LIN {X 0,Y 299.694,Z 797.286,A -85,B 0,C 180,E1 14832.527,E2 14832.527} C_VEL
LIN {X 0,Y 302.392,Z 789.527,A -85,B 0,C 180,E1 14828.672,E2 14828.672} C_VEL
LIN {X 0,Y 305.884,Z 780.362,A -85,B 0,C 180,E1 14825.061,E2 14825.061} C_VEL
LIN {X 0,Y 310.162,Z 769.656,A -85,B 0,C 180,E1 14821.65,E2 14821.65} C_VEL
LIN {X 0,Y 315.139,Z 757.152,A -85,B 0,C 180,E1 14818.433,E2 14818.433} C_VEL
LIN {X 0,Y 319.478,Z 746.033,A -85,B 0,C 180,E1 14816.053,E2 14816.053} C_VEL
LIN {X 0,Y 320.57,Z 741.155,A -85,B 0,C 180,E1 14814.994,E2 14814.994} C_VEL
LIN {X 0,Y 320.588,Z 728.797,A -85,B 0,C 180,E1 14812.148,E2 14812.148} C_VEL
LIN {X 0,Y 321.792,Z 723.281,A -85,B 0,C 180,E1 14811.202,E2 14811.202} C_VEL
LIN {X 0,Y 327.57,Z 706.668,A -85,B 0,C 180,E1 14808.986,E2 14808.986} C_VEL
LIN {X 0,Y 332.904,Z 689.548,A -85,B 0,C 180,E1 14807.126,E2 14807.126} C_VEL
LIN {X 0,Y 338.125,Z 670.498,A -85,B 0,C 180,E1 14805.452,E2 14805.452} C_VEL
LIN {X 0,Y 342.569,Z 651.293,A -85,B 0,C 180,E1 14804.112,E2 14804.112} C_VEL
LIN {X 0,Y 346.403,Z 631.027,A -85,B 0,C 180,E1 14803.025,E2 14803.025} C_VEL
LIN {X 0,Y 349.317,Z 610.319,A -85,B 0,C 180,E1 14802.217,E2 14802.217} C_VEL
LIN {X 0,Y 351.212,Z 589.58,A -85,B 0,C 180,E1 14801.664,E2 14801.664} C_VEL
LIN {X 0,Y 361.538,Z 397.142,A -85,B 0,C 180,E1 14797.851,E2 14797.851} C_VEL
LIN {X 0,Y 353.208,Z 382.377,A -85,B 0,C 180,E1 14795.383,E2 14795.383} C_VEL
LIN {X 0,Y 344.318,Z 367.821,A -85,B 0,C 180,E1 14792.446,E2 14792.446} C_VEL
LIN {X 0,Y 335.968,Z 355.363,A -85,B 0,C 180,E1 14789.313,E2 14789.313} C_VEL
LIN {X 0,Y 329.419,Z 346.302,A -85,B 0,C 180,E1 14786.499,E2 14786.499} C_VEL
LIN {X 0,Y 325.161,Z 340.597,A -85,B 0,C 180,E1 14784.43,E2 14784.43} C_VEL
LIN {X 0,Y 321.712,Z 336.158,A -85,B 0,C 180,E1 14782.571,E2 14782.571} C_VEL
LIN {X 0,Y 318.302,Z 331.619,A -85,B 0,C 180,E1 14780.503,E2 14780.503} C_VEL
LIN {X 0,Y 314.842,Z 327.176,A -85,B 0,C 180,E1 14778.085,E2 14778.085} C_VEL
LIN {X 0,Y 309.683,Z 320.807,A -85,B 0,C 180,E1 14773.442,E2 14773.442} C_VEL
LIN {X 0,Y 305.683,Z 315.348,A -85,B 0,C 180,E1 14766.197,E2 14766.197} C_VEL
LIN {X 0,Y 305.143,Z 314.738,A -85,B 0,C 180,E1 14761.127,E2 14761.127} C_VEL
LIN {X 0,Y 306.221,Z 315.739,A -85,B 0,C 180,E1 14756.818,E2 14756.818} C_VEL
LIN {X 0,Y 312.094,Z 322.032,A -85,B 0,C 180,E1 14749.385,E2 14749.385} C_VEL
LIN {X 0,Y 315.714,Z 326.528,A -85,B 0,C 180,E1 14746.447,E2 14746.447} C_VEL
LIN {X 0,Y 317.507,Z 328.292,A -85,B 0,C 180,E1 14745.222,E2 14745.222} C_VEL
LIN {X 0,Y 321.089,Z 332.723,A -85,B 0,C 180,E1 14742.98,E2 14742.98} C_VEL
LIN {X 0,Y 322.59,Z 334.467,A -85,B 0,C 180,E1 14742.131,E2 14742.131} C_VEL
LIN {X 0,Y 327.326,Z 340.382,A -85,B 0,C 180,E1 14739.668,E2 14739.668} C_VEL
LIN {X 0,Y 334.059,Z 349.029,A -85,B 0,C 180,E1 14736.636,E2 14736.636} C_VEL
LIN {X 0,Y 341.6,Z 359.524,A -85,B 0,C 180,E1 14733.677,E2 14733.677} C_VEL
LIN {X 0,Y 349.604,Z 371.289,A -85,B 0,C 180,E1 14730.91,E2 14730.91} C_VEL
LIN {X 0,Y 358.032,Z 384.909,A -85,B 0,C 180,E1 14728.284,E2 14728.284} C_VEL
LIN {X 0,Y 363.686,Z 394.863,A -85,B 0,C 180,E1 14726.65,E2 14726.65} C_VEL
LIN {X 0,Y 351.066,Z 599.637,A -85,B 0,C 180,E1 14722.328,E2 14722.328} C_VEL
LIN {X 0,Y 348.542,Z 622.55,A -85,B 0,C 180,E1 14721.656,E2 14721.656} C_VEL
LIN {X 0,Y 345.195,Z 643.809,A -85,B 0,C 180,E1 14720.786,E2 14720.786} C_VEL
LIN {X 0,Y 341.362,Z 663.255,A -85,B 0,C 180,E1 14719.728,E2 14719.728} C_VEL
LIN {X 0,Y 336.622,Z 683.448,A -85,B 0,C 180,E1 14718.331,E2 14718.331} C_VEL
LIN {X 0,Y 331.361,Z 702.998,A -85,B 0,C 180,E1 14716.65,E2 14716.65} C_VEL
LIN {X 0,Y 325.719,Z 721.816,A -85,B 0,C 180,E1 14714.663,E2 14714.663} C_VEL
LIN {X 0,Y 319.825,Z 739.772,A -85,B 0,C 180,E1 14712.333,E2 14712.333} C_VEL
LIN {X 0,Y 313.923,Z 756.677,A -85,B 0,C 180,E1 14709.686,E2 14709.686} C_VEL
LIN {X 0,Y 308.396,Z 772.066,A -85,B 0,C 180,E1 14706.794,E2 14706.794} C_VEL
LIN {X 0,Y 303.032,Z 786.885,A -85,B 0,C 180,E1 14703.436,E2 14703.436} C_VEL
LIN {X 0,Y 298.504,Z 799.576,A -85,B 0,C 180,E1 14699.939,E2 14699.939} C_VEL
LIN {X 0,Y 294.718,Z 810.947,A -85,B 0,C 180,E1 14696.169,E2 14696.169} C_VEL
LIN {X 0,Y 291.911,Z 820.502,A -85,B 0,C 180,E1 14692.345,E2 14692.345} C_VEL
LIN {X 0,Y 289.889,Z 828.607,A -85,B 0,C 180,E1 14688.292,E2 14688.292} C_VEL
LIN {X 0,Y 288.661,Z 835.273,A -85,B 0,C 180,E1 14684.032,E2 14684.032} C_VEL
LIN {X 0,Y 288.163,Z 840.012,A -85,B 0,C 180,E1 14679.99,E2 14679.99} C_VEL
LIN {X 0,Y 288.063,Z 842.936,A -85,B 0,C 180,E1 14676.177,E2 14676.177} C_VEL
LIN {X 0,Y 288.1,Z 844.57,A -85,B 0,C 180,E1 14672.387,E2 14672.387} C_VEL
LIN {X 0,Y 288.115,Z 844.72,A -85,B 0,C 180,E1 14668.807,E2 14668.807} C_VEL
LIN {X 0,Y 288.075,Z 843.64,A -85,B 0,C 180,E1 14665.022,E2 14665.022} C_VEL
LIN {X 0,Y 288.102,Z 841.035,A -85,B 0,C 180,E1 14661.217,E2 14661.217} C_VEL
LIN {X 0,Y 288.456,Z 836.889,A -85,B 0,C 180,E1 14657.183,E2 14657.183} C_VEL
LIN {X 0,Y 289.385,Z 831.018,A -85,B 0,C 180,E1 14653.129,E2 14653.129} C_VEL
LIN {X 0,Y 291.195,Z 823.048,A -85,B 0,C 180,E1 14648.868,E2 14648.868} C_VEL
LIN {X 0,Y 293.882,Z 813.618,A -85,B 0,C 180,E1 14644.832,E2 14644.832} C_VEL
LIN {X 0,Y 297.621,Z 802.16,A -85,B 0,C 180,E1 14640.849,E2 14640.849} C_VEL
LIN {X 0,Y 302.108,Z 789.305,A -85,B 0,C 180,E1 14637.207,E2 14637.207} C_VEL
LIN {X 0,Y 307.183,Z 775.278,A -85,B 0,C 180,E1 14633.905,E2 14633.905} C_VEL
LIN {X 0,Y 312.801,Z 759.732,A -85,B 0,C 180,E1 14630.855,E2 14630.855} C_VEL
LIN {X 0,Y 318.644,Z 743.198,A -85,B 0,C 180,E1 14628.168,E2 14628.168} C_VEL
LIN {X 0,Y 324.354,Z 725.842,A -85,B 0,C 180,E1 14625.841,E2 14625.841} C_VEL
LIN {X 0,Y 330.137,Z 706.989,A -85,B 0,C 180,E1 14623.755,E2 14623.755} C_VEL
LIN {X 0,Y 335.514,Z 687.59,A -85,B 0,C 180,E1 14622,E2 14622} C_VEL
LIN {X 0,Y 340.548,Z 666.776,A -85,B 0,C 180,E1 14620.5,E2 14620.5} C_VEL
LIN {X 0,Y 344.609,Z 646.553,A -85,B 0,C 180,E1 14619.362,E2 14619.362} C_VEL
LIN {X 0,Y 348.2,Z 624.526,A -85,B 0,C 180,E1 14618.425,E2 14618.425} C_VEL
LIN {X 0,Y 350.748,Z 602.835,A -85,B 0,C 180,E1 14617.76,E2 14617.76} C_VEL
LIN {X 0,Y 362.34,Z 415.076,A -85,B 0,C 180,E1 14613.778,E2 14613.778} C_VEL
LIN {X 0,Y 363.512,Z 394.465,A -85,B 0,C 180,E1 14613.327,E2 14613.327} C_VEL
LIN {X 0,Y 355.22,Z 380.343,A -85,B 0,C 180,E1 14610.91,E2 14610.91} C_VEL
LIN {X 0,Y 346.841,Z 367.12,A -85,B 0,C 180,E1 14608.214,E2 14608.214} C_VEL
LIN {X 0,Y 339.019,Z 355.984,A -85,B 0,C 180,E1 14605.411,E2 14605.411} C_VEL
LIN {X 0,Y 332.981,Z 347.726,A -85,B 0,C 180,E1 14602.976,E2 14602.976} C_VEL
LIN {X 0,Y 326.104,Z 338.74,A -85,B 0,C 180,E1 14599.803,E2 14599.803} C_VEL
LIN {X 0,Y 321.229,Z 332.843,A -85,B 0,C 180,E1 14597.199,E2 14597.199} C_VEL
LIN {X 0,Y 317.59,Z 328.472,A -85,B 0,C 180,E1 14594.96,E2 14594.96} C_VEL
LIN {X 0,Y 316.3,Z 326.994,A -85,B 0,C 180,E1 14594.087,E2 14594.087} C_VEL
LIN {X 0,Y 312.797,Z 323.164,A -85,B 0,C 180,E1 14591.43,E2 14591.43} C_VEL
LIN {X 0,Y 311.404,Z 321.292,A -85,B 0,C 180,E1 14590.171,E2 14590.171} C_VEL
LIN {X 0,Y 305.83,Z 315.283,A -85,B 0,C 180,E1 14582.811,E2 14582.811} C_VEL
LIN {X 0,Y 304.963,Z 314.593,A -85,B 0,C 180,E1 14577.557,E2 14577.557} C_VEL
LIN {X 0,Y 305.728,Z 315.381,A -85,B 0,C 180,E1 14573.05,E2 14573.05} C_VEL
LIN {X 0,Y 308.258,Z 319.618,A -85,B 0,C 180,E1 14567.828,E2 14567.828} C_VEL
LIN {X 0,Y 310.255,Z 321.599,A -85,B 0,C 180,E1 14565.632,E2 14565.632} C_VEL
LIN {X 0,Y 314.032,Z 326.159,A -85,B 0,C 180,E1 14562.298,E2 14562.298} C_VEL
LIN {X 0,Y 318.416,Z 331.744,A -85,B 0,C 180,E1 14559.216,E2 14559.216} C_VEL
LIN {X 0,Y 323.882,Z 338.999,A -85,B 0,C 180,E1 14556.049,E2 14556.049} C_VEL
LIN {X 0,Y 327.359,Z 343.584,A -85,B 0,C 180,E1 14554.296,E2 14554.296} C_VEL
LIN {X 0,Y 332.198,Z 350.191,A -85,B 0,C 180,E1 14552.093,E2 14552.093} C_VEL
LIN {X 0,Y 337.818,Z 358.315,A -85,B 0,C 180,E1 14549.79,E2 14549.79} C_VEL
LIN {X 0,Y 344.538,Z 368.286,A -85,B 0,C 180,E1 14547.331,E2 14547.331} C_VEL
LIN {X 0,Y 353.46,Z 382.878,A -85,B 0,C 180,E1 14544.407,E2 14544.407} C_VEL
LIN {X 0,Y 361.495,Z 397.193,A -85,B 0,C 180,E1 14542.032,E2 14542.032} C_VEL
LIN {X 0,Y 350.64,Z 596.622,A -85,B 0,C 180,E1 14538.077,E2 14538.077} C_VEL
LIN {X 0,Y 348.267,Z 617.827,A -85,B 0,C 180,E1 14537.42,E2 14537.42} C_VEL
LIN {X 0,Y 345.094,Z 637.899,A -85,B 0,C 180,E1 14536.533,E2 14536.533} C_VEL
LIN {X 0,Y 340.954,Z 658.356,A -85,B 0,C 180,E1 14535.326,E2 14535.326} C_VEL
LIN {X 0,Y 336.446,Z 676.774,A -85,B 0,C 180,E1 14533.94,E2 14533.94} C_VEL
LIN {X 0,Y 331.167,Z 695.218,A -85,B 0,C 180,E1 14532.202,E2 14532.202} C_VEL
LIN {X 0,Y 325.495,Z 712.561,A -85,B 0,C 180,E1 14530.17,E2 14530.17} C_VEL
LIN {X 0,Y 319.816,Z 728.387,A -85,B 0,C 180,E1 14527.902,E2 14527.902} C_VEL
LIN {X 0,Y 313.86,Z 743.787,A -85,B 0,C 180,E1 14525.211,E2 14525.211} C_VEL
LIN {X 0,Y 308.395,Z 757.265,A -85,B 0,C 180,E1 14522.34,E2 14522.34} C_VEL
LIN {X 0,Y 303.075,Z 770.006,A -85,B 0,C 180,E1 14519.009,E2 14519.009} C_VEL
LIN {X 0,Y 298.415,Z 781.102,A -85,B 0,C 180,E1 14515.395,E2 14515.395} C_VEL
LIN {X 0,Y 294.675,Z 790.399,A -85,B 0,C 180,E1 14511.61,E2 14511.61} C_VEL
LIN {X 0,Y 291.792,Z 798.237,A -85,B 0,C 180,E1 14507.55,E2 14507.55} C_VEL
LIN {X 0,Y 289.858,Z 804.348,A -85,B 0,C 180,E1 14503.362,E2 14503.362} C_VEL
LIN {X 0,Y 288.835,Z 808.554,A -85,B 0,C 180,E1 14499.363,E2 14499.363} C_VEL
LIN {X 0,Y 288.344,Z 811.162,A -85,B 0,C 180,E1 14495.372,E2 14495.372} C_VEL
LIN {X 0,Y 288.192,Z 812.368,A -85,B 0,C 180,E1 14491.392,E2 14491.392} C_VEL
LIN {X 0,Y 288.213,Z 812.225,A -85,B 0,C 180,E1 14487.415,E2 14487.415} C_VEL
LIN {X 0,Y 288.437,Z 810.589,A -85,B 0,C 180,E1 14483.432,E2 14483.432} C_VEL
LIN {X 0,Y 289.051,Z 807.519,A -85,B 0,C 180,E1 14479.436,E2 14479.436} C_VEL
LIN {X 0,Y 290.282,Z 802.961,A -85,B 0,C 180,E1 14475.437,E2 14475.437} C_VEL
LIN {X 0,Y 292.485,Z 796.391,A -85,B 0,C 180,E1 14471.25,E2 14471.25} C_VEL
LIN {X 0,Y 295.554,Z 788.243,A -85,B 0,C 180,E1 14467.316,E2 14467.316} C_VEL
LIN {X 0,Y 299.45,Z 778.638,A -85,B 0,C 180,E1 14463.636,E2 14463.636} C_VEL
LIN {X 0,Y 304.345,Z 766.977,A -85,B 0,C 180,E1 14460.043,E2 14460.043} C_VEL
LIN {X 0,Y 309.565,Z 754.489,A -85,B 0,C 180,E1 14456.918,E2 14456.918} C_VEL
LIN {X 0,Y 315.217,Z 740.609,A -85,B 0,C 180,E1 14454.07,E2 14454.07} C_VEL
LIN {X 0,Y 321.102,Z 725.141,A -85,B 0,C 180,E1 14451.483,E2 14451.483} C_VEL
LIN {X 0,Y 321.792,Z 723.281,A -85,B 0,C 180,E1 14451.202,E2 14451.202} C_VEL
LIN {X 0,Y 323.009,Z 717.705,A -85,B 0,C 180,E1 14450.286,E2 14450.286} C_VEL
LIN {X 0,Y 323.477,Z 703.653,A -85,B 0,C 180,E1 14447.742,E2 14447.742} C_VEL
LIN {X 0,Y 324.827,Z 697.456,A -85,B 0,C 180,E1 14446.922,E2 14446.922} C_VEL
LIN {X 0,Y 330.061,Z 680.098,A -85,B 0,C 180,E1 14445.227,E2 14445.227} C_VEL
LIN {X 0,Y 335.237,Z 660.245,A -85,B 0,C 180,E1 14443.677,E2 14443.677} C_VEL
LIN {X 0,Y 339.383,Z 641.044,A -85,B 0,C 180,E1 14442.503,E2 14442.503} C_VEL
LIN {X 0,Y 342.907,Z 620.295,A -85,B 0,C 180,E1 14441.545,E2 14441.545} C_VEL
LIN {X 0,Y 345.432,Z 599.009,A -85,B 0,C 180,E1 14440.861,E2 14440.861} C_VEL
LIN {X 0,Y 347.617,Z 564.108,A -85,B 0,C 180,E1 14440.124,E2 14440.124} C_VEL
LIN {X 0,Y 356.69,Z 400.719,A -85,B 0,C 180,E1 14436.861,E2 14436.861} C_VEL
LIN {X 0,Y 347.846,Z 385.024,A -85,B 0,C 180,E1 14434.092,E2 14434.092} C_VEL
LIN {X 0,Y 339.638,Z 371.67,A -85,B 0,C 180,E1 14431.207,E2 14431.207} C_VEL
LIN {X 0,Y 332.02,Z 360.277,A -85,B 0,C 180,E1 14428.167,E2 14428.167} C_VEL
LIN {X 0,Y 327.055,Z 353.249,A -85,B 0,C 180,E1 14425.924,E2 14425.924} C_VEL
LIN {X 0,Y 323.238,Z 347.975,A -85,B 0,C 180,E1 14424.002,E2 14424.002} C_VEL
LIN {X 0,Y 319.569,Z 343.174,A -85,B 0,C 180,E1 14421.956,E2 14421.956} C_VEL
LIN {X 0,Y 316.674,Z 339.189,A -85,B 0,C 180,E1 14420.131,E2 14420.131} C_VEL
LIN {X 0,Y 313.248,Z 334.655,A -85,B 0,C 180,E1 14417.652,E2 14417.652} C_VEL
LIN {X 0,Y 308.389,Z 328.55,A -85,B 0,C 180,E1 14413.118,E2 14413.118} C_VEL
LIN {X 0,Y 304.309,Z 323.127,A -85,B 0,C 180,E1 14405.846,E2 14405.846} C_VEL
LIN {X 0,Y 304.018,Z 322.706,A -85,B 0,C 180,E1 14400.566,E2 14400.566} C_VEL
LIN {X 0,Y 305.231,Z 323.746,A -85,B 0,C 180,E1 14396.808,E2 14396.808} C_VEL
LIN {X 0,Y 310.801,Z 329.875,A -85,B 0,C 180,E1 14389.622,E2 14389.622} C_VEL
LIN {X 0,Y 314.36,Z 334.318,A -85,B 0,C 180,E1 14386.668,E2 14386.668} C_VEL
LIN {X 0,Y 315.924,Z 335.945,A -85,B 0,C 180,E1 14385.568,E2 14385.568} C_VEL
LIN {X 0,Y 319.658,Z 340.529,A -85,B 0,C 180,E1 14383.182,E2 14383.182} C_VEL
LIN {X 0,Y 325.307,Z 347.74,A -85,B 0,C 180,E1 14380.099,E2 14380.099} C_VEL
LIN {X 0,Y 331.815,Z 356.306,A -85,B 0,C 180,E1 14377.079,E2 14377.079} C_VEL
LIN {X 0,Y 339.117,Z 366.695,A -85,B 0,C 180,E1 14374.128,E2 14374.128} C_VEL
LIN {X 0,Y 346.873,Z 378.361,A -85,B 0,C 180,E1 14371.366,E2 14371.366} C_VEL
LIN {X 0,Y 355.571,Z 392.721,A -85,B 0,C 180,E1 14368.583,E2 14368.583} C_VEL
LIN {X 0,Y 358.8,Z 398.776,A -85,B 0,C 180,E1 14367.606,E2 14367.606} C_VEL
LIN {X 0,Y 345.921,Z 600.369,A -85,B 0,C 180,E1 14363.328,E2 14363.328} C_VEL
LIN {X 0,Y 343.342,Z 622.749,A -85,B 0,C 180,E1 14362.664,E2 14362.664} C_VEL
LIN {X 0,Y 339.977,Z 643.47,A -85,B 0,C 180,E1 14361.815,E2 14361.815} C_VEL
LIN {X 0,Y 335.865,Z 663.645,A -85,B 0,C 180,E1 14360.713,E2 14360.713} C_VEL
LIN {X 0,Y 330.968,Z 683.704,A -85,B 0,C 180,E1 14359.31,E2 14359.31} C_VEL
LIN {X 0,Y 325.267,Z 703.98,A -85,B 0,C 180,E1 14357.538,E2 14357.538} C_VEL
LIN {X 0,Y 319.431,Z 722.613,A -85,B 0,C 180,E1 14355.532,E2 14355.532} C_VEL
LIN {X 0,Y 313.402,Z 740.196,A -85,B 0,C 180,E1 14353.208,E2 14353.208} C_VEL
LIN {X 0,Y 307.385,Z 756.647,A -85,B 0,C 180,E1 14350.582,E2 14350.582} C_VEL
LIN {X 0,Y 301.428,Z 772.4,A -85,B 0,C 180,E1 14347.555,E2 14347.555} C_VEL
LIN {X 0,Y 296.112,Z 786.365,A -85,B 0,C 180,E1 14344.325,E2 14344.325} C_VEL
LIN {X 0,Y 291.308,Z 799.073,A -85,B 0,C 180,E1 14340.757,E2 14340.757} C_VEL
LIN {X 0,Y 287.273,Z 810.458,A -85,B 0,C 180,E1 14336.901,E2 14336.901} C_VEL
LIN {X 0,Y 284.261,Z 820.023,A -85,B 0,C 180,E1 14332.981,E2 14332.981} C_VEL
LIN {X 0,Y 282.075,Z 828.134,A -85,B 0,C 180,E1 14328.817,E2 14328.817} C_VEL
LIN {X 0,Y 280.736,Z 834.809,A -85,B 0,C 180,E1 14324.436,E2 14324.436} C_VEL
LIN {X 0,Y 280.185,Z 839.555,A -85,B 0,C 180,E1 14320.278,E2 14320.278} C_VEL
LIN {X 0,Y 280.07,Z 842.484,A -85,B 0,C 180,E1 14316.354,E2 14316.354} C_VEL
LIN {X 0,Y 280.11,Z 844.121,A -85,B 0,C 180,E1 14312.455,E2 14312.455} C_VEL
LIN {X 0,Y 280.127,Z 844.271,A -85,B 0,C 180,E1 14308.773,E2 14308.773} C_VEL
LIN {X 0,Y 280.084,Z 843.265,A -85,B 0,C 180,E1 14305.085,E2 14305.085} C_VEL
LIN {X 0,Y 280.107,Z 840.751,A -85,B 0,C 180,E1 14301.171,E2 14301.171} C_VEL
LIN {X 0,Y 280.476,Z 836.685,A -85,B 0,C 180,E1 14297.022,E2 14297.022} C_VEL
LIN {X 0,Y 281.457,Z 830.871,A -85,B 0,C 180,E1 14292.852,E2 14292.852} C_VEL
LIN {X 0,Y 283.373,Z 822.996,A -85,B 0,C 180,E1 14288.473,E2 14288.473} C_VEL
LIN {X 0,Y 286.213,Z 813.66,A -85,B 0,C 180,E1 14284.329,E2 14284.329} C_VEL
LIN {X 0,Y 290.097,Z 802.382,A -85,B 0,C 180,E1 14280.29,E2 14280.29} C_VEL
LIN {X 0,Y 294.669,Z 789.997,A -85,B 0,C 180,E1 14276.655,E2 14276.655} C_VEL
LIN {X 0,Y 300.16,Z 775.621,A -85,B 0,C 180,E1 14273.16,E2 14273.16} C_VEL
LIN {X 0,Y 305.833,Z 760.74,A -85,B 0,C 180,E1 14270.151,E2 14270.151} C_VEL
LIN {X 0,Y 311.852,Z 744.401,A -85,B 0,C 180,E1 14267.43,E2 14267.43} C_VEL
LIN {X 0,Y 318.017,Z 726.59,A -85,B 0,C 180,E1 14264.977,E2 14264.977} C_VEL
LIN {X 0,Y 324.251,Z 707.133,A -85,B 0,C 180,E1 14262.788,E2 14262.788} C_VEL
LIN {X 0,Y 329.889,Z 687.58,A -85,B 0,C 180,E1 14261.003,E2 14261.003} C_VEL
LIN {X 0,Y 334.742,Z 668.225,A -85,B 0,C 180,E1 14259.591,E2 14259.591} C_VEL
LIN {X 0,Y 339.08,Z 647.706,A -85,B 0,C 180,E1 14258.408,E2 14258.408} C_VEL
LIN {X 0,Y 342.775,Z 626.229,A -85,B 0,C 180,E1 14257.471,E2 14257.471} C_VEL
LIN {X 0,Y 345.538,Z 604.181,A -85,B 0,C 180,E1 14256.775,E2 14256.775} C_VEL
LIN {X 0,Y 352.085,Z 502.283,A -85,B 0,C 180,E1 14254.573,E2 14254.573} C_VEL
LIN {X 0,Y 358.623,Z 398.228,A -85,B 0,C 180,E1 14252.364,E2 14252.364} C_VEL
LIN {X 0,Y 349.77,Z 383.094,A -85,B 0,C 180,E1 14249.639,E2 14249.639} C_VEL
LIN {X 0,Y 341.077,Z 369.503,A -85,B 0,C 180,E1 14246.648,E2 14246.648} C_VEL
LIN {X 0,Y 333.181,Z 358.323,A -85,B 0,C 180,E1 14243.57,E2 14243.57} C_VEL
LIN {X 0,Y 327.017,Z 350.061,A -85,B 0,C 180,E1 14240.82,E2 14240.82} C_VEL
LIN {X 0,Y 323.447,Z 345.423,A -85,B 0,C 180,E1 14239.034,E2 14239.034} C_VEL
LIN {X 0,Y 319.493,Z 340.384,A -85,B 0,C 180,E1 14236.826,E2 14236.826} C_VEL
LIN {X 0,Y 315.817,Z 335.815,A -85,B 0,C 180,E1 14234.484,E2 14234.484} C_VEL
LIN {X 0,Y 311.091,Z 330.377,A -85,B 0,C 180,E1 14230.837,E2 14230.837} C_VEL
LIN {X 0,Y 309.829,Z 328.884,A -85,B 0,C 180,E1 14229.66,E2 14229.66} C_VEL
LIN {X 0,Y 304.844,Z 323.243,A -85,B 0,C 180,E1 14222.82,E2 14222.82} C_VEL
LIN {X 0,Y 303.594,Z 322.469,A -85,B 0,C 180,E1 14217.735,E2 14217.735} C_VEL
LIN {X 0,Y 304.327,Z 323.219,A -85,B 0,C 180,E1 14213.207,E2 14213.207} C_VEL
LIN {X 0,Y 308.94,Z 329.307,A -85,B 0,C 180,E1 14205.952,E2 14205.952} C_VEL
LIN {X 0,Y 312.736,Z 333.971,A -85,B 0,C 180,E1 14202.51,E2 14202.51} C_VEL
LIN {X 0,Y 316.642,Z 339.18,A -85,B 0,C 180,E1 14199.675,E2 14199.675} C_VEL
LIN {X 0,Y 322.056,Z 346.494,A -85,B 0,C 180,E1 14196.439,E2 14196.439} C_VEL
LIN {X 0,Y 325.295,Z 350.873,A -85,B 0,C 180,E1 14194.756,E2 14194.756} C_VEL
LIN {X 0,Y 330.22,Z 357.733,A -85,B 0,C 180,E1 14192.451,E2 14192.451} C_VEL
LIN {X 0,Y 337.374,Z 368.235,A -85,B 0,C 180,E1 14189.501,E2 14189.501} C_VEL
LIN {X 0,Y 345.311,Z 380.88,A -85,B 0,C 180,E1 14186.622,E2 14186.622} C_VEL
LIN {X 0,Y 353.995,Z 395.883,A -85,B 0,C 180,E1 14183.82,E2 14183.82} C_VEL
LIN {X 0,Y 356.677,Z 401.111,A -85,B 0,C 180,E1 14183.002,E2 14183.002} C_VEL
LIN {X 0,Y 345.561,Z 596.845,A -85,B 0,C 180,E1 14179.095,E2 14179.095} C_VEL
LIN {X 0,Y 343.089,Z 618.172,A -85,B 0,C 180,E1 14178.431,E2 14178.431} C_VEL
LIN {X 0,Y 339.815,Z 638.167,A -85,B 0,C 180,E1 14177.542,E2 14177.542} C_VEL
LIN {X 0,Y 335.668,Z 658.048,A -85,B 0,C 180,E1 14176.37,E2 14176.37} C_VEL
LIN {X 0,Y 331.005,Z 676.58,A -85,B 0,C 180,E1 14174.977,E2 14174.977} C_VEL
LIN {X 0,Y 325.524,Z 695.074,A -85,B 0,C 180,E1 14173.23,E2 14173.23} C_VEL
LIN {X 0,Y 319.739,Z 712.182,A -85,B 0,C 180,E1 14171.224,E2 14171.224} C_VEL
LIN {X 0,Y 313.714,Z 728.395,A -85,B 0,C 180,E1 14168.892,E2 14168.892} C_VEL
LIN {X 0,Y 307.687,Z 743.404,A -85,B 0,C 180,E1 14166.257,E2 14166.257} C_VEL
LIN {X 0,Y 301.928,Z 757.015,A -85,B 0,C 180,E1 14163.347,E2 14163.347} C_VEL
LIN {X 0,Y 296.297,Z 769.823,A -85,B 0,C 180,E1 14159.961,E2 14159.961} C_VEL
LIN {X 0,Y 291.573,Z 780.481,A -85,B 0,C 180,E1 14156.473,E2 14156.473} C_VEL
LIN {X 0,Y 287.593,Z 789.793,A -85,B 0,C 180,E1 14152.699,E2 14152.699} C_VEL
LIN {X 0,Y 284.462,Z 797.695,A -85,B 0,C 180,E1 14148.654,E2 14148.654} C_VEL
LIN {X 0,Y 282.334,Z 803.839,A -85,B 0,C 180,E1 14144.562,E2 14144.562} C_VEL
LIN {X 0,Y 281.022,Z 808.446,A -85,B 0,C 180,E1 14140.247,E2 14140.247} C_VEL
LIN {X 0,Y 280.417,Z 811.296,A -85,B 0,C 180,E1 14136.14,E2 14136.14} C_VEL
LIN {X 0,Y 280.219,Z 812.755,A -85,B 0,C 180,E1 14132.045,E2 14132.045} C_VEL
LIN {X 0,Y 280.208,Z 812.787,A -85,B 0,C 180,E1 14128.16,E2 14128.16} C_VEL
LIN {X 0,Y 280.391,Z 811.461,A -85,B 0,C 180,E1 14124.064,E2 14124.064} C_VEL
LIN {X 0,Y 280.966,Z 808.746,A -85,B 0,C 180,E1 14119.958,E2 14119.958} C_VEL
LIN {X 0,Y 282.218,Z 804.215,A -85,B 0,C 180,E1 14115.641,E2 14115.641} C_VEL
LIN {X 0,Y 284.281,Z 798.206,A -85,B 0,C 180,E1 14111.547,E2 14111.547} C_VEL
LIN {X 0,Y 287.341,Z 790.46,A -85,B 0,C 180,E1 14107.496,E2 14107.496} C_VEL
LIN {X 0,Y 291.251,Z 781.313,A -85,B 0,C 180,E1 14103.715,E2 14103.715} C_VEL
LIN {X 0,Y 296.191,Z 770.165,A -85,B 0,C 180,E1 14100.027,E2 14100.027} C_VEL
LIN {X 0,Y 301.807,Z 757.391,A -85,B 0,C 180,E1 14096.638,E2 14096.638} C_VEL
LIN {X 0,Y 307.55,Z 743.853,A -85,B 0,C 180,E1 14093.724,E2 14093.724} C_VEL
LIN {X 0,Y 313.608,Z 728.837,A -85,B 0,C 180,E1 14091.072,E2 14091.072} C_VEL
LIN {X 0,Y 319.479,Z 713.142,A -85,B 0,C 180,E1 14088.794,E2 14088.794} C_VEL
LIN {X 0,Y 324.827,Z 697.456,A -85,B 0,C 180,E1 14086.922,E2 14086.922} C_VEL
LIN {X 0,Y 326.152,Z 691.249,A -85,B 0,C 180,E1 14086.133,E2 14086.133} C_VEL
LIN {X 0,Y 326.684,Z 675.586,A -85,B 0,C 180,E1 14083.918,E2 14083.918} C_VEL
LIN {X 0,Y 327.763,Z 668.933,A -85,B 0,C 180,E1 14083.253,E2 14083.253} C_VEL
LIN {X 0,Y 332.527,Z 649.214,A -85,B 0,C 180,E1 14081.912,E2 14081.912} C_VEL
LIN {X 0,Y 336.446,Z 629.158,A -85,B 0,C 180,E1 14080.868,E2 14080.868} C_VEL
LIN {X 0,Y 339.451,Z 608.763,A -85,B 0,C 180,E1 14080.086,E2 14080.086} C_VEL
LIN {X 0,Y 341.434,Z 587.116,A -85,B 0,C 180,E1 14079.53,E2 14079.53} C_VEL
LIN {X 0,Y 352.02,Z 404.613,A -85,B 0,C 180,E1 14075.871,E2 14075.871} C_VEL
LIN {X 0,Y 344.297,Z 390.709,A -85,B 0,C 180,E1 14073.339,E2 14073.339} C_VEL
LIN {X 0,Y 336.61,Z 377.939,A -85,B 0,C 180,E1 14070.527,E2 14070.527} C_VEL
LIN {X 0,Y 328.668,Z 365.741,A -85,B 0,C 180,E1 14067.199,E2 14067.199} C_VEL
LIN {X 0,Y 322.132,Z 356.327,A -85,B 0,C 180,E1 14063.992,E2 14063.992} C_VEL
LIN {X 0,Y 315.328,Z 347.018,A -85,B 0,C 180,E1 14059.93,E2 14059.93} C_VEL
LIN {X 0,Y 311.829,Z 342.431,A -85,B 0,C 180,E1 14057.35,E2 14057.35} C_VEL
LIN {X 0,Y 307.106,Z 336.297,A -85,B 0,C 180,E1 14052.791,E2 14052.791} C_VEL
LIN {X 0,Y 303.342,Z 331.091,A -85,B 0,C 180,E1 14045.865,E2 14045.865} C_VEL
LIN {X 0,Y 303.037,Z 330.646,A -85,B 0,C 180,E1 14040.568,E2 14040.568} C_VEL
LIN {X 0,Y 304.162,Z 331.618,A -85,B 0,C 180,E1 14036.985,E2 14036.985} C_VEL
LIN {X 0,Y 309.422,Z 337.559,A -85,B 0,C 180,E1 14029.951,E2 14029.951} C_VEL
LIN {X 0,Y 313.011,Z 342.108,A -85,B 0,C 180,E1 14026.892,E2 14026.892} C_VEL
LIN {X 0,Y 314.354,Z 343.593,A -85,B 0,C 180,E1 14025.918,E2 14025.918} C_VEL
LIN {X 0,Y 318.231,Z 348.336,A -85,B 0,C 180,E1 14023.387,E2 14023.387} C_VEL
LIN {X 0,Y 323.548,Z 355.45,A -85,B 0,C 180,E1 14020.41,E2 14020.41} C_VEL
LIN {X 0,Y 329.503,Z 363.439,A -85,B 0,C 180,E1 14017.569,E2 14017.569} C_VEL
LIN {X 0,Y 336.457,Z 373.55,A -85,B 0,C 180,E1 14014.664,E2 14014.664} C_VEL
LIN {X 0,Y 344.05,Z 385.248,A -85,B 0,C 180,E1 14011.867,E2 14011.867} C_VEL
LIN {X 0,Y 352.591,Z 399.715,A -85,B 0,C 180,E1 14009.047,E2 14009.047} C_VEL
LIN {X 0,Y 354.017,Z 402.668,A -85,B 0,C 180,E1 14008.589,E2 14008.589} C_VEL
LIN {X 0,Y 340.901,Z 600.896,A -85,B 0,C 180,E1 14004.364,E2 14004.364} C_VEL
LIN {X 0,Y 338.248,Z 622.979,A -85,B 0,C 180,E1 14003.702,E2 14003.702} C_VEL
LIN {X 0,Y 334.545,Z 644.767,A -85,B 0,C 180,E1 14002.794,E2 14002.794} C_VEL
LIN {X 0,Y 330.192,Z 665.328,A -85,B 0,C 180,E1 14001.652,E2 14001.652} C_VEL
LIN {X 0,Y 325.087,Z 685.18,A -85,B 0,C 180,E1 14000.228,E2 14000.228} C_VEL
LIN {X 0,Y 319.254,Z 704.967,A -85,B 0,C 180,E1 13998.46,E2 13998.46} C_VEL
LIN {X 0,Y 313.052,Z 723.831,A -85,B 0,C 180,E1 13996.38,E2 13996.38} C_VEL
LIN {X 0,Y 306.705,Z 741.616,A -85,B 0,C 180,E1 13993.976,E2 13993.976} C_VEL
LIN {X 0,Y 300.314,Z 758.185,A -85,B 0,C 180,E1 13991.239,E2 13991.239} C_VEL
LIN {X 0,Y 294.241,Z 773.413,A -85,B 0,C 180,E1 13988.202,E2 13988.202} C_VEL
LIN {X 0,Y 288.554,Z 787.588,A -85,B 0,C 180,E1 13984.793,E2 13984.793} C_VEL
LIN {X 0,Y 283.421,Z 800.59,A -85,B 0,C 180,E1 13980.991,E2 13980.991} C_VEL
LIN {X 0,Y 279.297,Z 811.594,A -85,B 0,C 180,E1 13977.041,E2 13977.041} C_VEL
LIN {X 0,Y 276.087,Z 821.262,A -85,B 0,C 180,E1 13972.799,E2 13972.799} C_VEL
LIN {X 0,Y 273.931,Z 829.127,A -85,B 0,C 180,E1 13968.514,E2 13968.514} C_VEL
LIN {X 0,Y 272.686,Z 835.162,A -85,B 0,C 180,E1 13964.221,E2 13964.221} C_VEL
LIN {X 0,Y 272.155,Z 839.792,A -85,B 0,C 180,E1 13959.729,E2 13959.729} C_VEL
LIN {X 0,Y 272.081,Z 842.4,A -85,B 0,C 180,E1 13955.906,E2 13955.906} C_VEL
LIN {X 0,Y 272.13,Z 843.75,A -85,B 0,C 180,E1 13951.895,E2 13951.895} C_VEL
LIN {X 0,Y 272.131,Z 843.773,A -85,B 0,C 180,E1 13948.316,E2 13948.316} C_VEL
LIN {X 0,Y 272.083,Z 842.513,A -85,B 0,C 180,E1 13944.306,E2 13944.306} C_VEL
LIN {X 0,Y 272.145,Z 839.95,A -85,B 0,C 180,E1 13940.484,E2 13940.484} C_VEL
LIN {X 0,Y 272.605,Z 835.687,A -85,B 0,C 180,E1 13936.208,E2 13936.208} C_VEL
LIN {X 0,Y 273.763,Z 829.754,A -85,B 0,C 180,E1 13931.915,E2 13931.915} C_VEL
LIN {X 0,Y 275.87,Z 821.929,A -85,B 0,C 180,E1 13927.549,E2 13927.549} C_VEL
LIN {X 0,Y 278.922,Z 812.633,A -85,B 0,C 180,E1 13923.38,E2 13923.38} C_VEL
LIN {X 0,Y 282.941,Z 801.766,A -85,B 0,C 180,E1 13919.413,E2 13919.413} C_VEL
LIN {X 0,Y 287.74,Z 789.485,A -85,B 0,C 180,E1 13915.742,E2 13915.742} C_VEL
LIN {X 0,Y 293.533,Z 775.088,A -85,B 0,C 180,E1 13912.185,E2 13912.185} C_VEL
LIN {X 0,Y 299.637,Z 759.824,A -85,B 0,C 180,E1 13909.069,E2 13909.069} C_VEL
LIN {X 0,Y 306.026,Z 743.257,A -85,B 0,C 180,E1 13906.291,E2 13906.291} C_VEL
LIN {X 0,Y 312.233,Z 725.973,A -85,B 0,C 180,E1 13903.905,E2 13903.905} C_VEL
LIN {X 0,Y 318.816,Z 706.147,A -85,B 0,C 180,E1 13901.672,E2 13901.672} C_VEL
LIN {X 0,Y 324.575,Z 686.81,A -85,B 0,C 180,E1 13899.912,E2 13899.912} C_VEL
LIN {X 0,Y 329.775,Z 666.697,A -85,B 0,C 180,E1 13898.451,E2 13898.451} C_VEL
LIN {X 0,Y 334.032,Z 646.942,A -85,B 0,C 180,E1 13897.327,E2 13897.327} C_VEL
LIN {X 0,Y 337.858,Z 625.124,A -85,B 0,C 180,E1 13896.387,E2 13896.387} C_VEL
LIN {X 0,Y 340.619,Z 603.314,A -85,B 0,C 180,E1 13895.706,E2 13895.706} C_VEL
LIN {X 0,Y 352.621,Z 422.147,A -85,B 0,C 180,E1 13891.826,E2 13891.826} C_VEL
LIN {X 0,Y 353.852,Z 402.085,A -85,B 0,C 180,E1 13891.382,E2 13891.382} C_VEL
LIN {X 0,Y 344.918,Z 386.714,A -85,B 0,C 180,E1 13888.48,E2 13888.48} C_VEL
LIN {X 0,Y 337.44,Z 375.081,A -85,B 0,C 180,E1 13885.774,E2 13885.774} C_VEL
LIN {X 0,Y 330.46,Z 364.924,A -85,B 0,C 180,E1 13882.926,E2 13882.926} C_VEL
LIN {X 0,Y 324.724,Z 357.088,A -85,B 0,C 180,E1 13880.267,E2 13880.267} C_VEL
LIN {X 0,Y 321.329,Z 352.595,A -85,B 0,C 180,E1 13878.505,E2 13878.505} C_VEL
LIN {X 0,Y 317.624,Z 347.786,A -85,B 0,C 180,E1 13876.364,E2 13876.364} C_VEL
LIN {X 0,Y 313.949,Z 342.947,A -85,B 0,C 180,E1 13873.913,E2 13873.913} C_VEL
LIN {X 0,Y 309.983,Z 338.536,A -85,B 0,C 180,E1 13870.782,E2 13870.782} C_VEL
LIN {X 0,Y 308.851,Z 336.896,A -85,B 0,C 180,E1 13869.691,E2 13869.691} C_VEL
LIN {X 0,Y 303.779,Z 331.127,A -85,B 0,C 180,E1 13862.641,E2 13862.641} C_VEL
LIN {X 0,Y 302.614,Z 330.421,A -85,B 0,C 180,E1 13857.348,E2 13857.348} C_VEL
LIN {X 0,Y 303.349,Z 331.239,A -85,B 0,C 180,E1 13853.185,E2 13853.185} C_VEL
LIN {X 0,Y 307.633,Z 337.016,A -85,B 0,C 180,E1 13846.275,E2 13846.275} C_VEL
LIN {X 0,Y 311.756,Z 342.411,A -85,B 0,C 180,E1 13842.453,E2 13842.453} C_VEL
LIN {X 0,Y 316.284,Z 348.471,A -85,B 0,C 180,E1 13839.215,E2 13839.215} C_VEL
LIN {X 0,Y 322.459,Z 356.867,A -85,B 0,C 180,E1 13835.644,E2 13835.644} C_VEL
LIN {X 0,Y 328.801,Z 366.062,A -85,B 0,C 180,E1 13832.567,E2 13832.567} C_VEL
LIN {X 0,Y 336.704,Z 378.181,A -85,B 0,C 180,E1 13829.285,E2 13829.285} C_VEL
LIN {X 0,Y 344.834,Z 391.678,A -85,B 0,C 180,E1 13826.339,E2 13826.339} C_VEL
LIN {X 0,Y 351.971,Z 404.788,A -85,B 0,C 180,E1 13824.004,E2 13824.004} C_VEL
LIN {X 0,Y 340.594,Z 597.062,A -85,B 0,C 180,E1 13820.143,E2 13820.143} C_VEL
LIN {X 0,Y 338.038,Z 618.39,A -85,B 0,C 180,E1 13819.477,E2 13819.477} C_VEL
LIN {X 0,Y 334.646,Z 638.433,A -85,B 0,C 180,E1 13818.583,E2 13818.583} C_VEL
LIN {X 0,Y 330.226,Z 658.858,A -85,B 0,C 180,E1 13817.369,E2 13817.369} C_VEL
LIN {X 0,Y 325.408,Z 677.271,A -85,B 0,C 180,E1 13815.97,E2 13815.97} C_VEL
LIN {X 0,Y 319.743,Z 695.725,A -85,B 0,C 180,E1 13814.212,E2 13814.212} C_VEL
LIN {X 0,Y 313.715,Z 712.864,A -85,B 0,C 180,E1 13812.177,E2 13812.177} C_VEL
LIN {X 0,Y 307.492,Z 728.941,A -85,B 0,C 180,E1 13809.833,E2 13809.833} C_VEL
LIN {X 0,Y 301.221,Z 743.922,A -85,B 0,C 180,E1 13807.164,E2 13807.164} C_VEL
LIN {X 0,Y 295.205,Z 757.511,A -85,B 0,C 180,E1 13804.21,E2 13804.21} C_VEL
LIN {X 0,Y 289.308,Z 770.313,A -85,B 0,C 180,E1 13800.762,E2 13800.762} C_VEL
LIN {X 0,Y 284.259,Z 781.132,A -85,B 0,C 180,E1 13797.138,E2 13797.138} C_VEL
LIN {X 0,Y 279.936,Z 790.698,A -85,B 0,C 180,E1 13793.134,E2 13793.134} C_VEL
LIN {X 0,Y 276.524,Z 798.826,A -85,B 0,C 180,E1 13788.772,E2 13788.772} C_VEL
LIN {X 0,Y 274.343,Z 804.784,A -85,B 0,C 180,E1 13784.564,E2 13784.564} C_VEL
LIN {X 0,Y 273.015,Z 809.288,A -85,B 0,C 180,E1 13780.124,E2 13780.124} C_VEL
LIN {X 0,Y 272.412,Z 811.958,A -85,B 0,C 180,E1 13775.899,E2 13775.899} C_VEL
LIN {X 0,Y 272.221,Z 813.244,A -85,B 0,C 180,E1 13771.684,E2 13771.684} C_VEL
LIN {X 0,Y 272.233,Z 813.194,A -85,B 0,C 180,E1 13767.685,E2 13767.685} C_VEL
LIN {X 0,Y 272.463,Z 811.699,A -85,B 0,C 180,E1 13763.468,E2 13763.468} C_VEL
LIN {X 0,Y 273.18,Z 808.618,A -85,B 0,C 180,E1 13759.029,E2 13759.029} C_VEL
LIN {X 0,Y 274.574,Z 804.158,A -85,B 0,C 180,E1 13754.797,E2 13754.797} C_VEL
LIN {X 0,Y 277.034,Z 797.661,A -85,B 0,C 180,E1 13750.388,E2 13750.388} C_VEL
LIN {X 0,Y 280.453,Z 789.611,A -85,B 0,C 180,E1 13746.243,E2 13746.243} C_VEL
LIN {X 0,Y 284.751,Z 780.135,A -85,B 0,C 180,E1 13742.388,E2 13742.388} C_VEL
LIN {X 0,Y 289.819,Z 769.264,A -85,B 0,C 180,E1 13738.825,E2 13738.825} C_VEL
LIN {X 0,Y 295.437,Z 757.125,A -85,B 0,C 180,E1 13735.586,E2 13735.586} C_VEL
LIN {X 0,Y 301.488,Z 743.463,A -85,B 0,C 180,E1 13732.635,E2 13732.635} C_VEL
LIN {X 0,Y 307.785,Z 728.387,A -85,B 0,C 180,E1 13729.969,E2 13729.969} C_VEL
LIN {X 0,Y 314.193,Z 711.758,A -85,B 0,C 180,E1 13727.575,E2 13727.575} C_VEL
LIN {X 0,Y 320.084,Z 694.891,A -85,B 0,C 180,E1 13725.597,E2 13725.597} C_VEL
LIN {X 0,Y 325.506,Z 677.226,A -85,B 0,C 180,E1 13723.921,E2 13723.921} C_VEL
LIN {X 0,Y 327.763,Z 668.933,A -85,B 0,C 180,E1 13723.253,E2 13723.253} C_VEL
LIN {X 0,Y 328.836,Z 663.118,A -85,B 0,C 180,E1 13722.717,E2 13722.717} C_VEL
LIN {X 0,Y 329.001,Z 645.229,A -85,B 0,C 180,E1 13720.728,E2 13720.728} C_VEL
LIN {X 0,Y 329.798,Z 638.124,A -85,B 0,C 180,E1 13720.21,E2 13720.21} C_VEL
LIN {X 0,Y 333.359,Z 617.472,A -85,B 0,C 180,E1 13719.303,E2 13719.303} C_VEL
LIN {X 0,Y 335.912,Z 596.493,A -85,B 0,C 180,E1 13718.657,E2 13718.657} C_VEL
LIN {X 0,Y 347.412,Z 408.429,A -85,B 0,C 180,E1 13714.84,E2 13714.84} C_VEL
LIN {X 0,Y 339.86,Z 394.672,A -85,B 0,C 180,E1 13712.224,E2 13712.224} C_VEL
LIN {X 0,Y 332.652,Z 382.655,A -85,B 0,C 180,E1 13709.435,E2 13709.435} C_VEL
LIN {X 0,Y 325.912,Z 372.169,A -85,B 0,C 180,E1 13706.463,E2 13706.463} C_VEL
LIN {X 0,Y 319.91,Z 363.316,A -85,B 0,C 180,E1 13703.387,E2 13703.387} C_VEL
LIN {X 0,Y 313.59,Z 354.457,A -85,B 0,C 180,E1 13699.463,E2 13699.463} C_VEL
LIN {X 0,Y 310.115,Z 349.609,A -85,B 0,C 180,E1 13696.772,E2 13696.772} C_VEL
LIN {X 0,Y 305.832,Z 344.051,A -85,B 0,C 180,E1 13692.461,E2 13692.461} C_VEL
LIN {X 0,Y 302.319,Z 338.985,A -85,B 0,C 180,E1 13685.695,E2 13685.695} C_VEL
LIN {X 0,Y 302.09,Z 338.606,A -85,B 0,C 180,E1 13680.38,E2 13680.38} C_VEL
LIN {X 0,Y 303.174,Z 339.626,A -85,B 0,C 180,E1 13676.976,E2 13676.976} C_VEL
LIN {X 0,Y 308.142,Z 345.396,A -85,B 0,C 180,E1 13670.192,E2 13670.192} C_VEL
LIN {X 0,Y 311.667,Z 349.899,A -85,B 0,C 180,E1 13667.117,E2 13667.117} C_VEL
LIN {X 0,Y 312.855,Z 351.332,A -85,B 0,C 180,E1 13666.226,E2 13666.226} C_VEL
LIN {X 0,Y 317.344,Z 357.151,A -85,B 0,C 180,E1 13663.245,E2 13663.245} C_VEL
LIN {X 0,Y 321.566,Z 362.804,A -85,B 0,C 180,E1 13660.851,E2 13660.851} C_VEL
LIN {X 0,Y 327.303,Z 370.709,A -85,B 0,C 180,E1 13658.024,E2 13658.024} C_VEL
LIN {X 0,Y 334.022,Z 380.71,A -85,B 0,C 180,E1 13655.13,E2 13655.13} C_VEL
LIN {X 0,Y 341.151,Z 391.958,A -85,B 0,C 180,E1 13652.415,E2 13652.415} C_VEL
LIN {X 0,Y 349.37,Z 406.216,A -85,B 0,C 180,E1 13649.607,E2 13649.607} C_VEL
LIN {X 0,Y 335.997,Z 601.435,A -85,B 0,C 180,E1 13645.43,E2 13645.43} C_VEL
LIN {X 0,Y 333.251,Z 623.331,A -85,B 0,C 180,E1 13644.767,E2 13644.767} C_VEL
LIN {X 0,Y 329.381,Z 645.253,A -85,B 0,C 180,E1 13643.846,E2 13643.846} C_VEL
LIN {X 0,Y 324.893,Z 665.676,A -85,B 0,C 180,E1 13642.703,E2 13642.703} C_VEL
LIN {X 0,Y 319.605,Z 685.531,A -85,B 0,C 180,E1 13641.268,E2 13641.268} C_VEL
LIN {X 0,Y 313.598,Z 705.128,A -85,B 0,C 180,E1 13639.499,E2 13639.499} C_VEL
LIN {X 0,Y 307.083,Z 724.137,A -85,B 0,C 180,E1 13637.378,E2 13637.378} C_VEL
LIN {X 0,Y 300.568,Z 741.65,A -85,B 0,C 180,E1 13634.981,E2 13634.981} C_VEL
LIN {X 0,Y 293.914,Z 758.159,A -85,B 0,C 180,E1 13632.21,E2 13632.21} C_VEL
LIN {X 0,Y 287.372,Z 773.765,A -85,B 0,C 180,E1 13629.031,E2 13629.031} C_VEL
LIN {X 0,Y 281.416,Z 787.842,A -85,B 0,C 180,E1 13625.549,E2 13625.549} C_VEL
LIN {X 0,Y 276.03,Z 800.787,A -85,B 0,C 180,E1 13621.655,E2 13621.655} C_VEL
LIN {X 0,Y 271.515,Z 812.188,A -85,B 0,C 180,E1 13617.407,E2 13617.407} C_VEL
LIN {X 0,Y 268.183,Z 821.643,A -85,B 0,C 180,E1 13613.045,E2 13613.045} C_VEL
LIN {X 0,Y 265.866,Z 829.63,A -85,B 0,C 180,E1 13608.415,E2 13608.415} C_VEL
LIN {X 0,Y 264.636,Z 835.515,A -85,B 0,C 180,E1 13603.993,E2 13603.993} C_VEL
LIN {X 0,Y 264.151,Z 839.682,A -85,B 0,C 180,E1 13599.587,E2 13599.587} C_VEL
LIN {X 0,Y 264.097,Z 842.335,A -85,B 0,C 180,E1 13595.318,E2 13595.318} C_VEL
LIN {X 0,Y 264.146,Z 843.352,A -85,B 0,C 180,E1 13591.518,E2 13591.518} C_VEL
LIN {X 0,Y 264.138,Z 843.273,A -85,B 0,C 180,E1 13587.831,E2 13587.831} C_VEL
LIN {X 0,Y 264.085,Z 841.815,A -85,B 0,C 180,E1 13583.697,E2 13583.697} C_VEL
LIN {X 0,Y 264.19,Z 839.132,A -85,B 0,C 180,E1 13579.735,E2 13579.735} C_VEL
LIN {X 0,Y 264.815,Z 834.406,A -85,B 0,C 180,E1 13575.123,E2 13575.123} C_VEL
LIN {X 0,Y 266.218,Z 828.287,A -85,B 0,C 180,E1 13570.701,E2 13570.701} C_VEL
LIN {X 0,Y 268.606,Z 820.321,A -85,B 0,C 180,E1 13566.296,E2 13566.296} C_VEL
LIN {X 0,Y 272.108,Z 810.52,A -85,B 0,C 180,E1 13561.945,E2 13561.945} C_VEL
LIN {X 0,Y 276.57,Z 799.343,A -85,B 0,C 180,E1 13557.899,E2 13557.899} C_VEL
LIN {X 0,Y 281.845,Z 786.787,A -85,B 0,C 180,E1 13554.174,E2 13554.174} C_VEL
LIN {X 0,Y 287.736,Z 772.807,A -85,B 0,C 180,E1 13550.771,E2 13550.771} C_VEL
LIN {X 0,Y 294.279,Z 757.125,A -85,B 0,C 180,E1 13547.62,E2 13547.62} C_VEL
LIN {X 0,Y 300.784,Z 740.902,A -85,B 0,C 180,E1 13544.925,E2 13544.925} C_VEL
LIN {X 0,Y 307.324,Z 723.31,A -85,B 0,C 180,E1 13542.534,E2 13542.534} C_VEL
LIN {X 0,Y 313.583,Z 704.952,A -85,B 0,C 180,E1 13540.497,E2 13540.497} C_VEL
LIN {X 0,Y 319.543,Z 685.466,A -85,B 0,C 180,E1 13538.741,E2 13538.741} C_VEL
LIN {X 0,Y 324.848,Z 665.524,A -85,B 0,C 180,E1 13537.3,E2 13537.3} C_VEL
LIN {X 0,Y 329.366,Z 644.919,A -85,B 0,C 180,E1 13536.15,E2 13536.15} C_VEL
LIN {X 0,Y 333.205,Z 623.039,A -85,B 0,C 180,E1 13535.235,E2 13535.235} C_VEL
LIN {X 0,Y 335.943,Z 600.95,A -85,B 0,C 180,E1 13534.571,E2 13534.571} C_VEL
LIN {X 0,Y 349.27,Z 406.145,A -85,B 0,C 180,E1 13530.401,E2 13530.401} C_VEL
LIN {X 0,Y 340.929,Z 391.695,A -85,B 0,C 180,E1 13527.557,E2 13527.557} C_VEL
LIN {X 0,Y 333.694,Z 380.289,A -85,B 0,C 180,E1 13524.802,E2 13524.802} C_VEL
LIN {X 0,Y 326.724,Z 369.896,A -85,B 0,C 180,E1 13521.78,E2 13521.78} C_VEL
LIN {X 0,Y 320.016,Z 360.652,A -85,B 0,C 180,E1 13518.394,E2 13518.394} C_VEL
LIN {X 0,Y 315.78,Z 355.182,A -85,B 0,C 180,E1 13515.895,E2 13515.895} C_VEL
LIN {X 0,Y 311.844,Z 350.053,A -85,B 0,C 180,E1 13513.158,E2 13513.158} C_VEL
LIN {X 0,Y 308.314,Z 345.749,A -85,B 0,C 180,E1 13510.18,E2 13510.18} C_VEL
LIN {X 0,Y 307.299,Z 344.491,A -85,B 0,C 180,E1 13509.174,E2 13509.174} C_VEL
LIN {X 0,Y 302.717,Z 339.013,A -85,B 0,C 180,E1 13502.461,E2 13502.461} C_VEL
LIN {X 0,Y 301.643,Z 338.368,A -85,B 0,C 180,E1 13497.15,E2 13497.15} C_VEL
LIN {X 0,Y 302.315,Z 339.124,A -85,B 0,C 180,E1 13493.352,E2 13493.352} C_VEL
LIN {X 0,Y 306.425,Z 344.898,A -85,B 0,C 180,E1 13486.493,E2 13486.493} C_VEL
LIN {X 0,Y 310.239,Z 349.981,A -85,B 0,C 180,E1 13482.849,E2 13482.849} C_VEL
LIN {X 0,Y 314.568,Z 355.937,A -85,B 0,C 180,E1 13479.641,E2 13479.641} C_VEL
LIN {X 0,Y 320.533,Z 364.297,A -85,B 0,C 180,E1 13476.076,E2 13476.076} C_VEL
LIN {X 0,Y 326.486,Z 373.106,A -85,B 0,C 180,E1 13473.097,E2 13473.097} C_VEL
LIN {X 0,Y 334.216,Z 385.274,A -85,B 0,C 180,E1 13469.778,E2 13469.778} C_VEL
LIN {X 0,Y 341.74,Z 398.08,A -85,B 0,C 180,E1 13466.955,E2 13466.955} C_VEL
LIN {X 0,Y 347.36,Z 408.698,A -85,B 0,C 180,E1 13465.028,E2 13465.028} C_VEL
LIN {X 0,Y 335.762,Z 597.074,A -85,B 0,C 180,E1 13461.226,E2 13461.226} C_VEL
LIN {X 0,Y 333.121,Z 618.462,A -85,B 0,C 180,E1 13460.559,E2 13460.559} C_VEL
LIN {X 0,Y 329.59,Z 638.695,A -85,B 0,C 180,E1 13459.657,E2 13459.657} C_VEL
LIN {X 0,Y 325.092,Z 658.839,A -85,B 0,C 180,E1 13458.459,E2 13458.459} C_VEL
LIN {X 0,Y 319.912,Z 677.962,A -85,B 0,C 180,E1 13456.998,E2 13456.998} C_VEL
LIN {X 0,Y 314.059,Z 696.37,A -85,B 0,C 180,E1 13455.23,E2 13455.23} C_VEL
LIN {X 0,Y 307.781,Z 713.553,A -85,B 0,C 180,E1 13453.166,E2 13453.166} C_VEL
LIN {X 0,Y 301.355,Z 729.486,A -85,B 0,C 180,E1 13450.814,E2 13450.814} C_VEL
LIN {X 0,Y 294.834,Z 744.435,A -85,B 0,C 180,E1 13448.111,E2 13448.111} C_VEL
LIN {X 0,Y 288.552,Z 758.005,A -85,B 0,C 180,E1 13445.113,E2 13445.113} C_VEL
LIN {X 0,Y 282.379,Z 770.803,A -85,B 0,C 180,E1 13441.603,E2 13441.603} C_VEL
LIN {X 0,Y 277.152,Z 781.434,A -85,B 0,C 180,E1 13437.968,E2 13437.968} C_VEL
LIN {X 0,Y 272.703,Z 790.727,A -85,B 0,C 180,E1 13434.014,E2 13434.014} C_VEL
LIN {X 0,Y 269.161,Z 798.617,A -85,B 0,C 180,E1 13429.757,E2 13429.757} C_VEL
LIN {X 0,Y 266.72,Z 804.755,A -85,B 0,C 180,E1 13425.435,E2 13425.435} C_VEL
LIN {X 0,Y 265.192,Z 809.355,A -85,B 0,C 180,E1 13420.866,E2 13420.866} C_VEL
LIN {X 0,Y 264.484,Z 812.196,A -85,B 0,C 180,E1 13416.512,E2 13416.512} C_VEL
LIN {X 0,Y 264.249,Z 813.651,A -85,B 0,C 180,E1 13412.168,E2 13412.168} C_VEL
LIN {X 0,Y 264.236,Z 813.683,A -85,B 0,C 180,E1 13408.048,E2 13408.048} C_VEL
LIN {X 0,Y 264.454,Z 812.36,A -85,B 0,C 180,E1 13403.705,E2 13403.705} C_VEL
LIN {X 0,Y 265.124,Z 809.653,A -85,B 0,C 180,E1 13399.351,E2 13399.351} C_VEL
LIN {X 0,Y 266.586,Z 805.124,A -85,B 0,C 180,E1 13394.78,E2 13394.78} C_VEL
LIN {X 0,Y 268.961,Z 799.125,A -85,B 0,C 180,E1 13390.454,E2 13390.454} C_VEL
LIN {X 0,Y 272.424,Z 791.39,A -85,B 0,C 180,E1 13386.189,E2 13386.189} C_VEL
LIN {X 0,Y 276.801,Z 782.26,A -85,B 0,C 180,E1 13382.228,E2 13382.228} C_VEL
LIN {X 0,Y 282.269,Z 771.134,A -85,B 0,C 180,E1 13378.383,E2 13378.383} C_VEL
LIN {X 0,Y 288.427,Z 758.37,A -85,B 0,C 180,E1 13374.87,E2 13374.87} C_VEL
LIN {X 0,Y 294.697,Z 744.872,A -85,B 0,C 180,E1 13371.868,E2 13371.868} C_VEL
LIN {X 0,Y 301.439,Z 729.466,A -85,B 0,C 180,E1 13369.074,E2 13369.074} C_VEL
LIN {X 0,Y 307.828,Z 713.646,A -85,B 0,C 180,E1 13366.738,E2 13366.738} C_VEL
LIN {X 0,Y 314.161,Z 696.324,A -85,B 0,C 180,E1 13364.659,E2 13364.659} C_VEL
LIN {X 0,Y 320.02,Z 677.904,A -85,B 0,C 180,E1 13362.892,E2 13362.892} C_VEL
LIN {X 0,Y 325,Z 659.591,A -85,B 0,C 180,E1 13361.487,E2 13361.487} C_VEL
LIN {X 0,Y 329.424,Z 640.054,A -85,B 0,C 180,E1 13360.309,E2 13360.309} C_VEL
LIN {X 0,Y 329.798,Z 638.124,A -85,B 0,C 180,E1 13360.21,E2 13360.21} C_VEL
LIN {X 0,Y 330.585,Z 630.92,A -85,B 0,C 180,E1 13359.719,E2 13359.719} C_VEL
LIN {X 0,Y 329.878,Z 612.939,A -85,B 0,C 180,E1 13358.164,E2 13358.164} C_VEL
LIN {X 0,Y 330.209,Z 605.509,A -85,B 0,C 180,E1 13357.791,E2 13357.791} C_VEL
LIN {X 0,Y 332.179,Z 583.872,A -85,B 0,C 180,E1 13357.261,E2 13357.261} C_VEL
LIN {X 0,Y 342.942,Z 412.34,A -85,B 0,C 180,E1 13353.795,E2 13353.795} C_VEL
LIN {X 0,Y 335.439,Z 398.551,A -85,B 0,C 180,E1 13351.043,E2 13351.043} C_VEL
LIN {X 0,Y 328.527,Z 387.02,A -85,B 0,C 180,E1 13348.197,E2 13348.197} C_VEL
LIN {X 0,Y 322.624,Z 377.665,A -85,B 0,C 180,E1 13345.419,E2 13345.419} C_VEL
LIN {X 0,Y 317.197,Z 369.606,A -85,B 0,C 180,E1 13342.47,E2 13342.47} C_VEL
LIN {X 0,Y 311.874,Z 361.892,A -85,B 0,C 180,E1 13338.991,E2 13338.991} C_VEL
LIN {X 0,Y 308.003,Z 356.476,A -85,B 0,C 180,E1 13335.825,E2 13335.825} C_VEL
LIN {X 0,Y 304.721,Z 351.936,A -85,B 0,C 180,E1 13332.315,E2 13332.315} C_VEL
LIN {X 0,Y 301.3,Z 346.881,A -85,B 0,C 180,E1 13325.523,E2 13325.523} C_VEL
LIN {X 0,Y 301.146,Z 346.567,A -85,B 0,C 180,E1 13320.191,E2 13320.191} C_VEL
LIN {X 0,Y 302.107,Z 347.498,A -85,B 0,C 180,E1 13317.155,E2 13317.155} C_VEL
LIN {X 0,Y 306.781,Z 353.078,A -85,B 0,C 180,E1 13310.527,E2 13310.527} C_VEL
LIN {X 0,Y 310.327,Z 357.689,A -85,B 0,C 180,E1 13307.345,E2 13307.345} C_VEL
LIN {X 0,Y 312.19,Z 360.348,A -85,B 0,C 180,E1 13305.913,E2 13305.913} C_VEL
LIN {X 0,Y 315.555,Z 364.599,A -85,B 0,C 180,E1 13303.668,E2 13303.668} C_VEL
LIN {X 0,Y 319.68,Z 370.272,A -85,B 0,C 180,E1 13301.255,E2 13301.255} C_VEL
LIN {X 0,Y 325.125,Z 377.973,A -85,B 0,C 180,E1 13298.486,E2 13298.486} C_VEL
LIN {X 0,Y 331.698,Z 388.012,A -85,B 0,C 180,E1 13295.562,E2 13295.562} C_VEL
LIN {X 0,Y 338.699,Z 399.354,A -85,B 0,C 180,E1 13292.818,E2 13292.818} C_VEL
LIN {X 0,Y 344.788,Z 410.381,A -85,B 0,C 180,E1 13290.638,E2 13290.638} C_VEL
LIN {X 0,Y 331.213,Z 601.983,A -85,B 0,C 180,E1 13286.527,E2 13286.527} C_VEL
LIN {X 0,Y 328.374,Z 623.69,A -85,B 0,C 180,E1 13285.864,E2 13285.864} C_VEL
LIN {X 0,Y 324.332,Z 645.743,A -85,B 0,C 180,E1 13284.931,E2 13284.931} C_VEL
LIN {X 0,Y 319.708,Z 666.006,A -85,B 0,C 180,E1 13283.789,E2 13283.789} C_VEL
LIN {X 0,Y 314.232,Z 685.886,A -85,B 0,C 180,E1 13282.344,E2 13282.344} C_VEL
LIN {X 0,Y 308.049,Z 705.292,A -85,B 0,C 180,E1 13280.577,E2 13280.577} C_VEL
LIN {X 0,Y 301.14,Z 724.628,A -85,B 0,C 180,E1 13278.391,E2 13278.391} C_VEL
LIN {X 0,Y 294.285,Z 742.245,A -85,B 0,C 180,E1 13275.936,E2 13275.936} C_VEL
LIN {X 0,Y 287.383,Z 758.658,A -85,B 0,C 180,E1 13273.129,E2 13273.129} C_VEL
LIN {X 0,Y 280.889,Z 773.393,A -85,B 0,C 180,E1 13270.065,E2 13270.065} C_VEL
LIN {X 0,Y 274.463,Z 787.807,A -85,B 0,C 180,E1 13266.426,E2 13266.426} C_VEL
LIN {X 0,Y 269,Z 800.22,A -85,B 0,C 180,E1 13262.612,E2 13262.612} C_VEL
LIN {X 0,Y 264.362,Z 811.161,A -85,B 0,C 180,E1 13258.46,E2 13258.46} C_VEL
LIN {X 0,Y 260.723,Z 820.739,A -85,B 0,C 180,E1 13253.985,E2 13253.985} C_VEL
LIN {X 0,Y 258.251,Z 828.516,A -85,B 0,C 180,E1 13249.448,E2 13249.448} C_VEL
LIN {X 0,Y 256.809,Z 834.508,A -85,B 0,C 180,E1 13244.89,E2 13244.89} C_VEL
LIN {X 0,Y 256.196,Z 838.88,A -85,B 0,C 180,E1 13240.342,E2 13240.342} C_VEL
LIN {X 0,Y 256.092,Z 841.497,A -85,B 0,C 180,E1 13236.276,E2 13236.276} C_VEL
LIN {X 0,Y 256.153,Z 842.853,A -85,B 0,C 180,E1 13232.013,E2 13232.013} C_VEL
LIN {X 0,Y 256.157,Z 842.901,A -85,B 0,C 180,E1 13228.434,E2 13228.434} C_VEL
LIN {X 0,Y 256.096,Z 841.731,A -85,B 0,C 180,E1 13224.174,E2 13224.174} C_VEL
LIN {X 0,Y 256.183,Z 839.036,A -85,B 0,C 180,E1 13219.885,E2 13219.885} C_VEL
LIN {X 0,Y 256.76,Z 834.758,A -85,B 0,C 180,E1 13215.338,E2 13215.338} C_VEL
LIN {X 0,Y 258.156,Z 828.815,A -85,B 0,C 180,E1 13210.78,E2 13210.78} C_VEL
LIN {X 0,Y 260.572,Z 821.129,A -85,B 0,C 180,E1 13206.241,E2 13206.241} C_VEL
LIN {X 0,Y 264.148,Z 811.653,A -85,B 0,C 180,E1 13201.762,E2 13201.762} C_VEL
LIN {X 0,Y 268.722,Z 800.777,A -85,B 0,C 180,E1 13197.603,E2 13197.603} C_VEL
LIN {X 0,Y 274.314,Z 788.047,A -85,B 0,C 180,E1 13193.661,E2 13193.661} C_VEL
LIN {X 0,Y 280.558,Z 774.031,A -85,B 0,C 180,E1 13190.099,E2 13190.099} C_VEL
LIN {X 0,Y 287.154,Z 759.072,A -85,B 0,C 180,E1 13186.965,E2 13186.965} C_VEL
LIN {X 0,Y 294.031,Z 742.691,A -85,B 0,C 180,E1 13184.152,E2 13184.152} C_VEL
LIN {X 0,Y 300.761,Z 725.432,A -85,B 0,C 180,E1 13181.728,E2 13181.728} C_VEL
LIN {X 0,Y 307.754,Z 705.932,A -85,B 0,C 180,E1 13179.503,E2 13179.503} C_VEL
LIN {X 0,Y 313.739,Z 687.314,A -85,B 0,C 180,E1 13177.783,E2 13177.783} C_VEL
LIN {X 0,Y 319.267,Z 667.319,A -85,B 0,C 180,E1 13176.314,E2 13176.314} C_VEL
LIN {X 0,Y 324.003,Z 646.879,A -85,B 0,C 180,E1 13175.139,E2 13175.139} C_VEL
LIN {X 0,Y 328.001,Z 625.529,A -85,B 0,C 180,E1 13174.215,E2 13174.215} C_VEL
LIN {X 0,Y 330.986,Z 603.448,A -85,B 0,C 180,E1 13173.521,E2 13173.521} C_VEL
LIN {X 0,Y 340.79,Z 465.235,A -85,B 0,C 180,E1 13170.527,E2 13170.527} C_VEL
LIN {X 0,Y 344.67,Z 410.085,A -85,B 0,C 180,E1 13169.357,E2 13169.357} C_VEL
LIN {X 0,Y 337.036,Z 396.658,A -85,B 0,C 180,E1 13166.612,E2 13166.612} C_VEL
LIN {X 0,Y 329.675,Z 384.893,A -85,B 0,C 180,E1 13163.646,E2 13163.646} C_VEL
LIN {X 0,Y 322.926,Z 374.862,A -85,B 0,C 180,E1 13160.527,E2 13160.527} C_VEL
LIN {X 0,Y 317.622,Z 367.472,A -85,B 0,C 180,E1 13157.684,E2 13157.684} C_VEL
LIN {X 0,Y 314.094,Z 362.716,A -85,B 0,C 180,E1 13155.509,E2 13155.509} C_VEL
LIN {X 0,Y 310.258,Z 357.636,A -85,B 0,C 180,E1 13152.753,E2 13152.753} C_VEL
LIN {X 0,Y 306.852,Z 353.277,A -85,B 0,C 180,E1 13149.755,E2 13149.755} C_VEL
LIN {X 0,Y 305.597,Z 351.942,A -85,B 0,C 180,E1 13148.466,E2 13148.466} C_VEL
LIN {X 0,Y 301.658,Z 346.901,A -85,B 0,C 180,E1 13142.279,E2 13142.279} C_VEL
LIN {X 0,Y 300.685,Z 346.332,A -85,B 0,C 180,E1 13136.759,E2 13136.759} C_VEL
LIN {X 0,Y 301.336,Z 347.153,A -85,B 0,C 180,E1 13133.331,E2 13133.331} C_VEL
LIN {X 0,Y 305.123,Z 352.582,A -85,B 0,C 180,E1 13126.835,E2 13126.835} C_VEL
LIN {X 0,Y 308.837,Z 357.737,A -85,B 0,C 180,E1 13123.156,E2 13123.156} C_VEL
LIN {X 0,Y 312.896,Z 363.445,A -85,B 0,C 180,E1 13120.055,E2 13120.055} C_VEL
LIN {X 0,Y 318.556,Z 371.59,A -85,B 0,C 180,E1 13116.557,E2 13116.557} C_VEL
LIN {X 0,Y 324.284,Z 380.292,A -85,B 0,C 180,E1 13113.591,E2 13113.591} C_VEL
LIN {X 0,Y 331.651,Z 392.193,A -85,B 0,C 180,E1 13110.318,E2 13110.318} C_VEL
LIN {X 0,Y 338.799,Z 404.705,A -85,B 0,C 180,E1 13107.54,E2 13107.54} C_VEL
LIN {X 0,Y 342.866,Z 412.603,A -85,B 0,C 180,E1 13106.079,E2 13106.079} C_VEL
LIN {X 0,Y 331.035,Z 597.282,A -85,B 0,C 180,E1 13102.336,E2 13102.336} C_VEL
LIN {X 0,Y 328.308,Z 618.676,A -85,B 0,C 180,E1 13101.668,E2 13101.668} C_VEL
LIN {X 0,Y 324.655,Z 638.952,A -85,B 0,C 180,E1 13100.763,E2 13100.763} C_VEL
LIN {X 0,Y 319.966,Z 659.264,A -85,B 0,C 180,E1 13099.553,E2 13099.553} C_VEL
LIN {X 0,Y 314.835,Z 677.671,A -85,B 0,C 180,E1 13098.148,E2 13098.148} C_VEL
LIN {X 0,Y 308.88,Z 695.813,A -85,B 0,C 180,E1 13096.41,E2 13096.41} C_VEL
LIN {X 0,Y 302.441,Z 712.952,A -85,B 0,C 180,E1 13094.362,E2 13094.362} C_VEL
LIN {X 0,Y 295.786,Z 728.946,A -85,B 0,C 180,E1 13092.012,E2 13092.012} C_VEL
LIN {X 0,Y 288.967,Z 744.048,A -85,B 0,C 180,E1 13089.285,E2 13089.285} C_VEL
LIN {X 0,Y 282.367,Z 757.734,A -85,B 0,C 180,E1 13086.251,E2 13086.251} C_VEL
LIN {X 0,Y 275.846,Z 770.613,A -85,B 0,C 180,E1 13082.688,E2 13082.688} C_VEL
LIN {X 0,Y 270.294,Z 781.358,A -85,B 0,C 180,E1 13078.985,E2 13078.985} C_VEL
LIN {X 0,Y 265.315,Z 791.195,A -85,B 0,C 180,E1 13074.727,E2 13074.727} C_VEL
LIN {X 0,Y 261.551,Z 799.077,A -85,B 0,C 180,E1 13070.357,E2 13070.357} C_VEL
LIN {X 0,Y 258.938,Z 805.212,A -85,B 0,C 180,E1 13065.911,E2 13065.911} C_VEL
LIN {X 0,Y 257.287,Z 809.809,A -85,B 0,C 180,E1 13061.204,E2 13061.204} C_VEL
LIN {X 0,Y 256.522,Z 812.646,A -85,B 0,C 180,E1 13056.715,E2 13056.715} C_VEL
LIN {X 0,Y 256.263,Z 814.099,A -85,B 0,C 180,E1 13052.236,E2 13052.236} C_VEL
LIN {X 0,Y 256.245,Z 814.152,A -85,B 0,C 180,E1 13048.211,E2 13048.211} C_VEL
LIN {X 0,Y 256.467,Z 812.916,A -85,B 0,C 180,E1 13043.733,E2 13043.733} C_VEL
LIN {X 0,Y 257.165,Z 810.291,A -85,B 0,C 180,E1 13039.244,E2 13039.244} C_VEL
LIN {X 0,Y 258.695,Z 805.817,A -85,B 0,C 180,E1 13034.533,E2 13034.533} C_VEL
LIN {X 0,Y 261.185,Z 799.918,A -85,B 0,C 180,E1 13030.081,E2 13030.081} C_VEL
LIN {X 0,Y 265.023,Z 791.854,A -85,B 0,C 180,E1 13025.481,E2 13025.481} C_VEL
LIN {X 0,Y 269.651,Z 782.731,A -85,B 0,C 180,E1 13021.425,E2 13021.425} C_VEL
LIN {X 0,Y 275.404,Z 771.615,A -85,B 0,C 180,E1 13017.5,E2 13017.5} C_VEL
LIN {X 0,Y 281.849,Z 758.858,A -85,B 0,C 180,E1 13013.923,E2 13013.923} C_VEL
LIN {X 0,Y 288.395,Z 745.38,A -85,B 0,C 180,E1 13010.878,E2 13010.878} C_VEL
LIN {X 0,Y 295.405,Z 730.002,A -85,B 0,C 180,E1 13008.052,E2 13008.052} C_VEL
LIN {X 0,Y 302.035,Z 714.222,A -85,B 0,C 180,E1 13005.695,E2 13005.695} C_VEL
LIN {X 0,Y 308.587,Z 696.941,A -85,B 0,C 180,E1 13003.602,E2 13003.602} C_VEL
LIN {X 0,Y 314.64,Z 678.578,A -85,B 0,C 180,E1 13001.826,E2 13001.826} C_VEL
LIN {X 0,Y 319.78,Z 660.38,A -85,B 0,C 180,E1 13000.418,E2 13000.418} C_VEL
LIN {X 0,Y 324.343,Z 641.029,A -85,B 0,C 180,E1 12999.239,E2 12999.239} C_VEL
LIN {X 0,Y 328.177,Z 620.365,A -85,B 0,C 180,E1 12998.29,E2 12998.29} C_VEL
LIN {X 0,Y 330.209,Z 605.509,A -85,B 0,C 180,E1 12997.791,E2 12997.791} C_VEL
LIN {X 0,Y 330.517,Z 598.003,A -85,B 0,C 180,E1 12997.444,E2 12997.444} C_VEL
LIN {X 0,Y 328.422,Z 578.299,A -85,B 0,C 180,E1 12996.111,E2 12996.111} C_VEL
LIN {X 0,Y 328.403,Z 571.788,A -85,B 0,C 180,E1 12995.869,E2 12995.869} C_VEL
LIN {X 0,Y 338.573,Z 416.229,A -85,B 0,C 180,E1 12992.713,E2 12992.713} C_VEL
LIN {X 0,Y 331.345,Z 402.937,A -85,B 0,C 180,E1 12989.911,E2 12989.911} C_VEL
LIN {X 0,Y 325.354,Z 392.756,A -85,B 0,C 180,E1 12987.301,E2 12987.301} C_VEL
LIN {X 0,Y 319.21,Z 382.775,A -85,B 0,C 180,E1 12984.226,E2 12984.226} C_VEL
LIN {X 0,Y 313.756,Z 374.494,A -85,B 0,C 180,E1 12981.009,E2 12981.009} C_VEL
LIN {X 0,Y 310.058,Z 369.183,A -85,B 0,C 180,E1 12978.423,E2 12978.423} C_VEL
LIN {X 0,Y 306.544,Z 364.072,A -85,B 0,C 180,E1 12975.417,E2 12975.417} C_VEL
LIN {X 0,Y 303.461,Z 359.691,A -85,B 0,C 180,E1 12971.981,E2 12971.981} C_VEL
LIN {X 0,Y 300.282,Z 354.779,A -85,B 0,C 180,E1 12965.35,E2 12965.35} C_VEL
LIN {X 0,Y 300.21,Z 354.528,A -85,B 0,C 180,E1 12960,E2 12960} C_VEL
LIN {X 0,Y 301.119,Z 355.505,A -85,B 0,C 180,E1 12957.145,E2 12957.145} C_VEL
LIN {X 0,Y 305.515,Z 360.913,A -85,B 0,C 180,E1 12950.772,E2 12950.772} C_VEL
LIN {X 0,Y 308.993,Z 365.479,A -85,B 0,C 180,E1 12947.574,E2 12947.574} C_VEL
LIN {X 0,Y 313.854,Z 372.151,A -85,B 0,C 180,E1 12944.052,E2 12944.052} C_VEL
LIN {X 0,Y 317.81,Z 377.738,A -85,B 0,C 180,E1 12941.663,E2 12941.663} C_VEL
LIN {X 0,Y 322.963,Z 385.232,A -85,B 0,C 180,E1 12938.954,E2 12938.954} C_VEL
LIN {X 0,Y 330.354,Z 396.75,A -85,B 0,C 180,E1 12935.598,E2 12935.598} C_VEL
LIN {X 0,Y 337.904,Z 409.706,A -85,B 0,C 180,E1 12932.605,E2 12932.605} C_VEL
LIN {X 0,Y 340.327,Z 414.513,A -85,B 0,C 180,E1 12931.699,E2 12931.699} C_VEL
LIN {X 0,Y 326.563,Z 602.429,A -85,B 0,C 180,E1 12927.659,E2 12927.659} C_VEL
LIN {X 0,Y 323.599,Z 624.181,A -85,B 0,C 180,E1 12926.989,E2 12926.989} C_VEL
LIN {X 0,Y 319.565,Z 645.492,A -85,B 0,C 180,E1 12926.088,E2 12926.088} C_VEL
LIN {X 0,Y 314.956,Z 665.193,A -85,B 0,C 180,E1 12924.987,E2 12924.987} C_VEL
LIN {X 0,Y 309.41,Z 684.763,A -85,B 0,C 180,E1 12923.574,E2 12923.574} C_VEL
LIN {X 0,Y 303.192,Z 703.807,A -85,B 0,C 180,E1 12921.859,E2 12921.859} C_VEL
LIN {X 0,Y 296.449,Z 722.253,A -85,B 0,C 180,E1 12919.811,E2 12919.811} C_VEL
LIN {X 0,Y 289.343,Z 739.869,A -85,B 0,C 180,E1 12917.394,E2 12917.394} C_VEL
LIN {X 0,Y 282.294,Z 756.024,A -85,B 0,C 180,E1 12914.672,E2 12914.672} C_VEL
LIN {X 0,Y 275.063,Z 771.851,A -85,B 0,C 180,E1 12911.419,E2 12911.419} C_VEL
LIN {X 0,Y 268.376,Z 786.114,A -85,B 0,C 180,E1 12907.831,E2 12907.831} C_VEL
LIN {X 0,Y 262.283,Z 799.126,A -85,B 0,C 180,E1 12903.794,E2 12903.794} C_VEL
LIN {X 0,Y 257.309,Z 810.136,A -85,B 0,C 180,E1 12899.57,E2 12899.57} C_VEL
LIN {X 0,Y 253.165,Z 820.263,A -85,B 0,C 180,E1 12894.748,E2 12894.748} C_VEL
LIN {X 0,Y 250.485,Z 828.048,A -85,B 0,C 180,E1 12890.077,E2 12890.077} C_VEL
LIN {X 0,Y 248.907,Z 834.045,A -85,B 0,C 180,E1 12885.374,E2 12885.374} C_VEL
LIN {X 0,Y 248.217,Z 838.465,A -85,B 0,C 180,E1 12880.622,E2 12880.622} C_VEL
LIN {X 0,Y 248.099,Z 841.168,A -85,B 0,C 180,E1 12876.247,E2 12876.247} C_VEL
LIN {X 0,Y 248.166,Z 842.43,A -85,B 0,C 180,E1 12871.847,E2 12871.847} C_VEL
LIN {X 0,Y 248.166,Z 842.427,A -85,B 0,C 180,E1 12868.153,E2 12868.153} C_VEL
LIN {X 0,Y 248.099,Z 841.155,A -85,B 0,C 180,E1 12863.753,E2 12863.753} C_VEL
LIN {X 0,Y 248.219,Z 838.446,A -85,B 0,C 180,E1 12859.375,E2 12859.375} C_VEL
LIN {X 0,Y 248.962,Z 833.749,A -85,B 0,C 180,E1 12854.391,E2 12854.391} C_VEL
LIN {X 0,Y 250.609,Z 827.639,A -85,B 0,C 180,E1 12849.648,E2 12849.648} C_VEL
LIN {X 0,Y 253.327,Z 819.794,A -85,B 0,C 180,E1 12845.02,E2 12845.02} C_VEL
LIN {X 0,Y 257.306,Z 810.084,A -85,B 0,C 180,E1 12840.43,E2 12840.43} C_VEL
LIN {X 0,Y 262.302,Z 799.003,A -85,B 0,C 180,E1 12836.185,E2 12836.185} C_VEL
LIN {X 0,Y 268.359,Z 786.061,A -85,B 0,C 180,E1 12832.173,E2 12832.173} C_VEL
LIN {X 0,Y 275.054,Z 771.756,A -85,B 0,C 180,E1 12828.58,E2 12828.58} C_VEL
LIN {X 0,Y 282.282,Z 755.908,A -85,B 0,C 180,E1 12825.326,E2 12825.326} C_VEL
LIN {X 0,Y 289.33,Z 739.724,A -85,B 0,C 180,E1 12822.603,E2 12822.603} C_VEL
LIN {X 0,Y 296.435,Z 722.092,A -85,B 0,C 180,E1 12820.186,E2 12820.186} C_VEL
LIN {X 0,Y 303.175,Z 703.61,A -85,B 0,C 180,E1 12818.136,E2 12818.136} C_VEL
LIN {X 0,Y 309.721,Z 683.393,A -85,B 0,C 180,E1 12816.333,E2 12816.333} C_VEL
LIN {X 0,Y 315.171,Z 663.936,A -85,B 0,C 180,E1 12814.949,E2 12814.949} C_VEL
LIN {X 0,Y 320.034,Z 642.888,A -85,B 0,C 180,E1 12813.796,E2 12813.796} C_VEL
LIN {X 0,Y 323.924,Z 621.445,A -85,B 0,C 180,E1 12812.927,E2 12812.927} C_VEL
LIN {X 0,Y 326.839,Z 598.065,A -85,B 0,C 180,E1 12812.248,E2 12812.248} C_VEL
LIN {X 0,Y 340.196,Z 414.069,A -85,B 0,C 180,E1 12808.289,E2 12808.289} C_VEL
LIN {X 0,Y 333.231,Z 401.686,A -85,B 0,C 180,E1 12805.646,E2 12805.646} C_VEL
LIN {X 0,Y 326.496,Z 390.798,A -85,B 0,C 180,E1 12802.792,E2 12802.792} C_VEL
LIN {X 0,Y 319.615,Z 380.246,A -85,B 0,C 180,E1 12799.413,E2 12799.413} C_VEL
LIN {X 0,Y 315.282,Z 374.264,A -85,B 0,C 180,E1 12796.963,E2 12796.963} C_VEL
LIN {X 0,Y 312.287,Z 370.104,A -85,B 0,C 180,E1 12795.031,E2 12795.031} C_VEL
LIN {X 0,Y 308.688,Z 365.213,A -85,B 0,C 180,E1 12792.343,E2 12792.343} C_VEL
LIN {X 0,Y 305.323,Z 360.648,A -85,B 0,C 180,E1 12789.233,E2 12789.233} C_VEL
LIN {X 0,Y 300.681,Z 354.859,A -85,B 0,C 180,E1 12782.287,E2 12782.287} C_VEL
LIN {X 0,Y 299.702,Z 354.26,A -85,B 0,C 180,E1 12776.94,E2 12776.94} C_VEL
LIN {X 0,Y 300.308,Z 355.039,A -85,B 0,C 180,E1 12773.5,E2 12773.5} C_VEL
LIN {X 0,Y 303.915,Z 360.436,A -85,B 0,C 180,E1 12767.072,E2 12767.072} C_VEL
LIN {X 0,Y 307.345,Z 365.302,A -85,B 0,C 180,E1 12763.559,E2 12763.559} C_VEL
LIN {X 0,Y 311.292,Z 371.035,A -85,B 0,C 180,E1 12760.436,E2 12760.436} C_VEL
LIN {X 0,Y 316.601,Z 378.882,A -85,B 0,C 180,E1 12757.044,E2 12757.044} C_VEL
LIN {X 0,Y 322.018,Z 387.333,A -85,B 0,C 180,E1 12754.135,E2 12754.135} C_VEL
LIN {X 0,Y 329.021,Z 398.946,A -85,B 0,C 180,E1 12750.907,E2 12750.907} C_VEL
LIN {X 0,Y 335.855,Z 411.245,A -85,B 0,C 180,E1 12748.151,E2 12748.151} C_VEL
LIN {X 0,Y 338.489,Z 416.523,A -85,B 0,C 180,E1 12747.158,E2 12747.158} C_VEL
LIN {X 0,Y 326.454,Z 597.284,A -85,B 0,C 180,E1 12743.482,E2 12743.482} C_VEL
LIN {X 0,Y 323.648,Z 618.696,A -85,B 0,C 180,E1 12742.816,E2 12742.816} C_VEL
LIN {X 0,Y 319.997,Z 638.472,A -85,B 0,C 180,E1 12741.941,E2 12741.941} C_VEL
LIN {X 0,Y 315.134,Z 659.032,A -85,B 0,C 180,E1 12740.727,E2 12740.727} C_VEL
LIN {X 0,Y 309.804,Z 677.637,A -85,B 0,C 180,E1 12739.312,E2 12739.312} C_VEL
LIN {X 0,Y 303.555,Z 696.07,A -85,B 0,C 180,E1 12737.544,E2 12737.544} C_VEL
LIN {X 0,Y 296.76,Z 713.535,A -85,B 0,C 180,E1 12735.445,E2 12735.445} C_VEL
LIN {X 0,Y 289.86,Z 729.485,A -85,B 0,C 180,E1 12733.076,E2 12733.076} C_VEL
LIN {X 0,Y 282.77,Z 744.56,A -85,B 0,C 180,E1 12730.32,E2 12730.32} C_VEL
LIN {X 0,Y 275.891,Z 758.234,A -85,B 0,C 180,E1 12727.244,E2 12727.244} C_VEL
LIN {X 0,Y 269.065,Z 771.101,A -85,B 0,C 180,E1 12723.619,E2 12723.619} C_VEL
LIN {X 0,Y 263.229,Z 781.833,A -85,B 0,C 180,E1 12719.84,E2 12719.84} C_VEL
LIN {X 0,Y 257.969,Z 791.66,A -85,B 0,C 180,E1 12715.481,E2 12715.481} C_VEL
LIN {X 0,Y 253.969,Z 799.538,A -85,B 0,C 180,E1 12710.993,E2 12710.993} C_VEL
LIN {X 0,Y 251.152,Z 805.718,A -85,B 0,C 180,E1 12706.373,E2 12706.373} C_VEL
LIN {X 0,Y 249.395,Z 810.264,A -85,B 0,C 180,E1 12701.563,E2 12701.563} C_VEL
LIN {X 0,Y 248.561,Z 813.097,A -85,B 0,C 180,E1 12696.931,E2 12696.931} C_VEL
LIN {X 0,Y 248.277,Z 814.548,A -85,B 0,C 180,E1 12692.308,E2 12692.308} C_VEL
LIN {X 0,Y 248.259,Z 814.6,A -85,B 0,C 180,E1 12688.154,E2 12688.154} C_VEL
LIN {X 0,Y 248.501,Z 813.366,A -85,B 0,C 180,E1 12683.532,E2 12683.532} C_VEL
LIN {X 0,Y 249.261,Z 810.743,A -85,B 0,C 180,E1 12678.899,E2 12678.899} C_VEL
LIN {X 0,Y 250.912,Z 806.271,A -85,B 0,C 180,E1 12674.041,E2 12674.041} C_VEL
LIN {X 0,Y 253.581,Z 800.376,A -85,B 0,C 180,E1 12669.457,E2 12669.457} C_VEL
LIN {X 0,Y 257.665,Z 792.318,A -85,B 0,C 180,E1 12664.733,E2 12664.733} C_VEL
LIN {X 0,Y 262.556,Z 783.203,A -85,B 0,C 180,E1 12660.578,E2 12660.578} C_VEL
LIN {X 0,Y 268.607,Z 772.094,A -85,B 0,C 180,E1 12656.571,E2 12656.571} C_VEL
LIN {X 0,Y 275.355,Z 759.345,A -85,B 0,C 180,E1 12652.932,E2 12652.932} C_VEL
LIN {X 0,Y 282.181,Z 745.886,A -85,B 0,C 180,E1 12649.844,E2 12649.844} C_VEL
LIN {X 0,Y 289.468,Z 730.536,A -85,B 0,C 180,E1 12646.987,E2 12646.987} C_VEL
LIN {X 0,Y 296.347,Z 714.797,A -85,B 0,C 180,E1 12644.612,E2 12644.612} C_VEL
LIN {X 0,Y 303.121,Z 697.546,A -85,B 0,C 180,E1 12642.506,E2 12642.506} C_VEL
LIN {X 0,Y 309.085,Z 680.13,A -85,B 0,C 180,E1 12640.803,E2 12640.803} C_VEL
LIN {X 0,Y 314.675,Z 661.168,A -85,B 0,C 180,E1 12639.314,E2 12639.314} C_VEL
LIN {X 0,Y 319.379,Z 642.003,A -85,B 0,C 180,E1 12638.136,E2 12638.136} C_VEL
LIN {X 0,Y 323.402,Z 621.114,A -85,B 0,C 180,E1 12637.169,E2 12637.169} C_VEL
LIN {X 0,Y 326.28,Z 599.813,A -85,B 0,C 180,E1 12636.482,E2 12636.482} C_VEL
LIN {X 0,Y 328.403,Z 571.788,A -85,B 0,C 180,E1 12635.869,E2 12635.869} C_VEL
LIN {X 0,Y 328.323,Z 564.213,A -85,B 0,C 180,E1 12635.566,E2 12635.566} C_VEL
LIN {X 0,Y 326.222,Z 544.467,A -85,B 0,C 180,E1 12634.239,E2 12634.239} C_VEL
LIN {X 0,Y 326.284,Z 537.951,A -85,B 0,C 180,E1 12634.001,E2 12634.001} C_VEL
LIN {X 0,Y 334.324,Z 420.268,A -85,B 0,C 180,E1 12631.611,E2 12631.611} C_VEL
LIN {X 0,Y 327.3,Z 407.065,A -85,B 0,C 180,E1 12628.711,E2 12628.711} C_VEL
LIN {X 0,Y 320.746,Z 395.866,A -85,B 0,C 180,E1 12625.628,E2 12625.628} C_VEL
LIN {X 0,Y 315.983,Z 388.254,A -85,B 0,C 180,E1 12623.053,E2 12623.053} C_VEL
LIN {X 0,Y 311.844,Z 381.683,A -85,B 0,C 180,E1 12620.456,E2 12620.456} C_VEL
LIN {X 0,Y 308.391,Z 376.605,A -85,B 0,C 180,E1 12617.94,E2 12617.94} C_VEL
LIN {X 0,Y 305.194,Z 371.776,A -85,B 0,C 180,E1 12615.097,E2 12615.097} C_VEL
LIN {X 0,Y 302.212,Z 367.446,A -85,B 0,C 180,E1 12611.644,E2 12611.644} C_VEL
LIN {X 0,Y 299.267,Z 362.68,A -85,B 0,C 180,E1 12605.176,E2 12605.176} C_VEL
LIN {X 0,Y 299.322,Z 362.515,A -85,B 0,C 180,E1 12599.618,E2 12599.618} C_VEL
LIN {X 0,Y 300.131,Z 363.518,A -85,B 0,C 180,E1 12597.136,E2 12597.136} C_VEL
LIN {X 0,Y 304.253,Z 368.748,A -85,B 0,C 180,E1 12591.02,E2 12591.02} C_VEL
LIN {X 0,Y 308.201,Z 374.133,A -85,B 0,C 180,E1 12587.351,E2 12587.351} C_VEL
LIN {X 0,Y 312.365,Z 380.007,A -85,B 0,C 180,E1 12584.308,E2 12584.308} C_VEL
LIN {X 0,Y 316.026,Z 385.312,A -85,B 0,C 180,E1 12582.033,E2 12582.033} C_VEL
LIN {X 0,Y 320.99,Z 392.756,A -85,B 0,C 180,E1 12579.344,E2 12579.344} C_VEL
LIN {X 0,Y 327.769,Z 403.62,A -85,B 0,C 180,E1 12576.16,E2 12576.16} C_VEL
LIN {X 0,Y 334.941,Z 416.266,A -85,B 0,C 180,E1 12573.208,E2 12573.208} C_VEL
LIN {X 0,Y 335.991,Z 418.58,A -85,B 0,C 180,E1 12572.789,E2 12572.789} C_VEL
LIN {X 0,Y 322.074,Z 602.571,A -85,B 0,C 180,E1 12568.83,E2 12568.83} C_VEL
LIN {X 0,Y 318.995,Z 624.419,A -85,B 0,C 180,E1 12568.157,E2 12568.157} C_VEL
LIN {X 0,Y 314.767,Z 645.99,A -85,B 0,C 180,E1 12567.241,E2 12567.241} C_VEL
LIN {X 0,Y 309.699,Z 666.672,A -85,B 0,C 180,E1 12566.068,E2 12566.068} C_VEL
LIN {X 0,Y 303.836,Z 686.602,A -85,B 0,C 180,E1 12564.608,E2 12564.608} C_VEL
LIN {X 0,Y 297.296,Z 705.627,A -85,B 0,C 180,E1 12562.849,E2 12562.849} C_VEL
LIN {X 0,Y 289.783,Z 725.071,A -85,B 0,C 180,E1 12560.611,E2 12560.611} C_VEL
LIN {X 0,Y 282.556,Z 742.15,A -85,B 0,C 180,E1 12558.179,E2 12558.179} C_VEL
LIN {X 0,Y 275.025,Z 758.613,A -85,B 0,C 180,E1 12555.294,E2 12555.294} C_VEL
LIN {X 0,Y 267.552,Z 774.04,A -85,B 0,C 180,E1 12551.955,E2 12551.955} C_VEL
LIN {X 0,Y 260.5,Z 788.263,A -85,B 0,C 180,E1 12548.166,E2 12548.166} C_VEL
LIN {X 0,Y 254.499,Z 800.454,A -85,B 0,C 180,E1 12544.18,E2 12544.18} C_VEL
LIN {X 0,Y 249.136,Z 811.812,A -85,B 0,C 180,E1 12539.579,E2 12539.579} C_VEL
LIN {X 0,Y 245.136,Z 821.073,A -85,B 0,C 180,E1 12534.841,E2 12534.841} C_VEL
LIN {X 0,Y 242.318,Z 828.875,A -85,B 0,C 180,E1 12529.776,E2 12529.776} C_VEL
LIN {X 0,Y 240.795,Z 834.626,A -85,B 0,C 180,E1 12524.918,E2 12524.918} C_VEL
LIN {X 0,Y 240.198,Z 838.488,A -85,B 0,C 180,E1 12520.311,E2 12520.311} C_VEL
LIN {X 0,Y 240.122,Z 841.096,A -85,B 0,C 180,E1 12515.496,E2 12515.496} C_VEL
LIN {X 0,Y 240.183,Z 842.032,A -85,B 0,C 180,E1 12511.431,E2 12511.431} C_VEL
LIN {X 0,Y 240.165,Z 841.901,A -85,B 0,C 180,E1 12507.375,E2 12507.375} C_VEL
LIN {X 0,Y 240.117,Z 840.333,A -85,B 0,C 180,E1 12502.824,E2 12502.824} C_VEL
LIN {X 0,Y 240.314,Z 837.428,A -85,B 0,C 180,E1 12498.237,E2 12498.237} C_VEL
LIN {X 0,Y 241.211,Z 832.74,A -85,B 0,C 180,E1 12493.381,E2 12493.381} C_VEL
LIN {X 0,Y 243.23,Z 826.115,A -85,B 0,C 180,E1 12488.287,E2 12488.287} C_VEL
LIN {X 0,Y 246.386,Z 818.03,A -85,B 0,C 180,E1 12483.488,E2 12483.488} C_VEL
LIN {X 0,Y 250.855,Z 807.976,A -85,B 0,C 180,E1 12478.792,E2 12478.792} C_VEL
LIN {X 0,Y 256.373,Z 796.516,A -85,B 0,C 180,E1 12474.473,E2 12474.473} C_VEL
LIN {X 0,Y 262.735,Z 783.708,A -85,B 0,C 180,E1 12470.542,E2 12470.542} C_VEL
LIN {X 0,Y 269.748,Z 769.484,A -85,B 0,C 180,E1 12467,E2 12467} C_VEL
LIN {X 0,Y 277.174,Z 753.794,A -85,B 0,C 180,E1 12463.826,E2 12463.826} C_VEL
LIN {X 0,Y 284.855,Z 736.643,A -85,B 0,C 180,E1 12461.006,E2 12461.006} C_VEL
LIN {X 0,Y 292.203,Z 718.925,A -85,B 0,C 180,E1 12458.64,E2 12458.64} C_VEL
LIN {X 0,Y 299.075,Z 700.464,A -85,B 0,C 180,E1 12456.646,E2 12456.646} C_VEL
LIN {X 0,Y 305.223,Z 681.713,A -85,B 0,C 180,E1 12455.022,E2 12455.022} C_VEL
LIN {X 0,Y 311.142,Z 660.696,A -85,B 0,C 180,E1 12453.574,E2 12453.574} C_VEL
LIN {X 0,Y 316.036,Z 639.701,A -85,B 0,C 180,E1 12452.466,E2 12452.466} C_VEL
LIN {X 0,Y 319.971,Z 617.762,A -85,B 0,C 180,E1 12451.625,E2 12451.625} C_VEL
LIN {X 0,Y 322.571,Z 595.842,A -85,B 0,C 180,E1 12451.021,E2 12451.021} C_VEL
LIN {X 0,Y 335.84,Z 418.112,A -85,B 0,C 180,E1 12447.193,E2 12447.193} C_VEL
LIN {X 0,Y 329.328,Z 406.411,A -85,B 0,C 180,E1 12444.578,E2 12444.578} C_VEL
LIN {X 0,Y 322.283,Z 394.797,A -85,B 0,C 180,E1 12441.379,E2 12441.379} C_VEL
LIN {X 0,Y 316.24,Z 385.705,A -85,B 0,C 180,E1 12438.193,E2 12438.193} C_VEL
LIN {X 0,Y 313.135,Z 381.226,A -85,B 0,C 180,E1 12436.319,E2 12436.319} C_VEL
LIN {X 0,Y 310.503,Z 377.487,A -85,B 0,C 180,E1 12434.546,E2 12434.546} C_VEL
LIN {X 0,Y 307.134,Z 372.789,A -85,B 0,C 180,E1 12431.93,E2 12431.93} C_VEL
LIN {X 0,Y 303.634,Z 367.969,A -85,B 0,C 180,E1 12428.521,E2 12428.521} C_VEL
LIN {X 0,Y 299.63,Z 362.748,A -85,B 0,C 180,E1 12422.103,E2 12422.103} C_VEL
LIN {X 0,Y 298.737,Z 362.218,A -85,B 0,C 180,E1 12416.738,E2 12416.738} C_VEL
LIN {X 0,Y 299.333,Z 363.065,A -85,B 0,C 180,E1 12413.478,E2 12413.478} C_VEL
LIN {X 0,Y 302.642,Z 368.141,A -85,B 0,C 180,E1 12407.405,E2 12407.405} C_VEL
LIN {X 0,Y 305.968,Z 373.05,A -85,B 0,C 180,E1 12403.873,E2 12403.873} C_VEL
LIN {X 0,Y 309.703,Z 378.622,A -85,B 0,C 180,E1 12400.822,E2 12400.822} C_VEL
LIN {X 0,Y 314.737,Z 386.298,A -85,B 0,C 180,E1 12397.492,E2 12397.492} C_VEL
LIN {X 0,Y 319.781,Z 394.373,A -85,B 0,C 180,E1 12394.686,E2 12394.686} C_VEL
LIN {X 0,Y 326.52,Z 405.862,A -85,B 0,C 180,E1 12391.464,E2 12391.464} C_VEL
LIN {X 0,Y 332.997,Z 417.873,A -85,B 0,C 180,E1 12388.755,E2 12388.755} C_VEL
LIN {X 0,Y 334.221,Z 420.57,A -85,B 0,C 180,E1 12388.262,E2 12388.262} C_VEL
LIN {X 0,Y 321.988,Z 597.481,A -85,B 0,C 180,E1 12384.656,E2 12384.656} C_VEL
LIN {X 0,Y 319.088,Z 618.936,A -85,B 0,C 180,E1 12383.989,E2 12383.989} C_VEL
LIN {X 0,Y 315.322,Z 638.725,A -85,B 0,C 180,E1 12383.115,E2 12383.115} C_VEL
LIN {X 0,Y 310.464,Z 658.71,A -85,B 0,C 180,E1 12381.943,E2 12381.943} C_VEL
LIN {X 0,Y 304.989,Z 677.353,A -85,B 0,C 180,E1 12380.536,E2 12380.536} C_VEL
LIN {X 0,Y 298.499,Z 695.915,A -85,B 0,C 180,E1 12378.761,E2 12378.761} C_VEL
LIN {X 0,Y 291.638,Z 713.047,A -85,B 0,C 180,E1 12376.71,E2 12376.71} C_VEL
LIN {X 0,Y 284.038,Z 730.027,A -85,B 0,C 180,E1 12374.185,E2 12374.185} C_VEL
LIN {X 0,Y 276.669,Z 745.07,A -85,B 0,C 180,E1 12371.401,E2 12371.401} C_VEL
LIN {X 0,Y 269.502,Z 758.729,A -85,B 0,C 180,E1 12368.284,E2 12368.284} C_VEL
LIN {X 0,Y 262.343,Z 771.617,A -85,B 0,C 180,E1 12364.589,E2 12364.589} C_VEL
LIN {X 0,Y 256.227,Z 782.308,A -85,B 0,C 180,E1 12360.742,E2 12360.742} C_VEL
LIN {X 0,Y 250.67,Z 792.127,A -85,B 0,C 180,E1 12356.279,E2 12356.279} C_VEL
LIN {X 0,Y 246.419,Z 799.997,A -85,B 0,C 180,E1 12351.668,E2 12351.668} C_VEL
LIN {X 0,Y 243.349,Z 806.29,A -85,B 0,C 180,E1 12346.795,E2 12346.795} C_VEL
LIN {X 0,Y 241.445,Z 810.912,A -85,B 0,C 180,E1 12341.707,E2 12341.707} C_VEL
LIN {X 0,Y 240.574,Z 813.653,A -85,B 0,C 180,E1 12336.922,E2 12336.922} C_VEL
LIN {X 0,Y 240.286,Z 815.017,A -85,B 0,C 180,E1 12332.146,E2 12332.146} C_VEL
LIN {X 0,Y 240.279,Z 815.028,A -85,B 0,C 180,E1 12327.854,E2 12327.854} C_VEL
LIN {X 0,Y 240.564,Z 813.71,A -85,B 0,C 180,E1 12323.077,E2 12323.077} C_VEL
LIN {X 0,Y 241.425,Z 811.012,A -85,B 0,C 180,E1 12318.292,E2 12318.292} C_VEL
LIN {X 0,Y 243.277,Z 806.468,A -85,B 0,C 180,E1 12313.261,E2 12313.261} C_VEL
LIN {X 0,Y 246.183,Z 800.499,A -85,B 0,C 180,E1 12308.56,E2 12308.56} C_VEL
LIN {X 0,Y 250.593,Z 792.342,A -85,B 0,C 180,E1 12303.713,E2 12303.713} C_VEL
LIN {X 0,Y 255.824,Z 783.122,A -85,B 0,C 180,E1 12299.464,E2 12299.464} C_VEL
LIN {X 0,Y 262.037,Z 772.3,A -85,B 0,C 180,E1 12295.508,E2 12295.508} C_VEL
LIN {X 0,Y 268.947,Z 759.83,A -85,B 0,C 180,E1 12291.894,E2 12291.894} C_VEL
LIN {X 0,Y 276.063,Z 746.391,A -85,B 0,C 180,E1 12288.764,E2 12288.764} C_VEL
LIN {X 0,Y 283.893,Z 730.526,A -85,B 0,C 180,E1 12285.787,E2 12285.787} C_VEL
LIN {X 0,Y 291.03,Z 714.741,A -85,B 0,C 180,E1 12283.403,E2 12283.403} C_VEL
LIN {X 0,Y 298.061,Z 697.414,A -85,B 0,C 180,E1 12281.288,E2 12281.288} C_VEL
LIN {X 0,Y 304.526,Z 679.034,A -85,B 0,C 180,E1 12279.506,E2 12279.506} C_VEL
LIN {X 0,Y 309.995,Z 660.83,A -85,B 0,C 180,E1 12278.096,E2 12278.096} C_VEL
LIN {X 0,Y 315.001,Z 640.76,A -85,B 0,C 180,E1 12276.883,E2 12276.883} C_VEL
LIN {X 0,Y 319.011,Z 620.246,A -85,B 0,C 180,E1 12275.954,E2 12275.954} C_VEL
LIN {X 0,Y 321.967,Z 598.743,A -85,B 0,C 180,E1 12275.273,E2 12275.273} C_VEL
LIN {X 0,Y 325.374,Z 551.554,A -85,B 0,C 180,E1 12274.278,E2 12274.278} C_VEL
LIN {X 0,Y 326.284,Z 537.951,A -85,B 0,C 180,E1 12274.001,E2 12274.001} C_VEL
LIN {X 0,Y 326.295,Z 530.376,A -85,B 0,C 180,E1 12273.705,E2 12273.705} C_VEL
LIN {X 0,Y 324.422,Z 510.65,A -85,B 0,C 180,E1 12272.349,E2 12272.349} C_VEL
LIN {X 0,Y 324.493,Z 504.139,A -85,B 0,C 180,E1 12272.099,E2 12272.099} C_VEL
LIN {X 0,Y 330.136,Z 424.235,A -85,B 0,C 180,E1 12270.459,E2 12270.459} C_VEL
LIN {X 0,Y 323.817,Z 412.196,A -85,B 0,C 180,E1 12267.691,E2 12267.691} C_VEL
LIN {X 0,Y 317.209,Z 400.629,A -85,B 0,C 180,E1 12264.368,E2 12264.368} C_VEL
LIN {X 0,Y 311.73,Z 391.737,A -85,B 0,C 180,E1 12261.103,E2 12261.103} C_VEL
LIN {X 0,Y 306.973,Z 384.308,A -85,B 0,C 180,E1 12257.633,E2 12257.633} C_VEL
LIN {X 0,Y 303.76,Z 379.374,A -85,B 0,C 180,E1 12254.682,E2 12254.682} C_VEL
LIN {X 0,Y 301.111,Z 375.33,A -85,B 0,C 180,E1 12251.493,E2 12251.493} C_VEL
LIN {X 0,Y 298.295,Z 370.636,A -85,B 0,C 180,E1 12245.193,E2 12245.193} C_VEL
LIN {X 0,Y 298.302,Z 370.432,A -85,B 0,C 180,E1 12239.808,E2 12239.808} C_VEL
LIN {X 0,Y 299.07,Z 371.392,A -85,B 0,C 180,E1 12237.318,E2 12237.318} C_VEL
LIN {X 0,Y 302.92,Z 376.43,A -85,B 0,C 180,E1 12231.363,E2 12231.363} C_VEL
LIN {X 0,Y 306.747,Z 381.854,A -85,B 0,C 180,E1 12227.673,E2 12227.673} C_VEL
LIN {X 0,Y 310.618,Z 387.45,A -85,B 0,C 180,E1 12224.743,E2 12224.743} C_VEL
LIN {X 0,Y 314.4,Z 393.094,A -85,B 0,C 180,E1 12222.32,E2 12222.32} C_VEL
LIN {X 0,Y 320.274,Z 402.182,A -85,B 0,C 180,E1 12219.104,E2 12219.104} C_VEL
LIN {X 0,Y 327.423,Z 414.351,A -85,B 0,C 180,E1 12215.75,E2 12215.75} C_VEL
LIN {X 0,Y 331.78,Z 422.617,A -85,B 0,C 180,E1 12213.907,E2 12213.907} C_VEL
LIN {X 0,Y 317.742,Z 602.502,A -85,B 0,C 180,E1 12210.039,E2 12210.039} C_VEL
LIN {X 0,Y 314.57,Z 624.401,A -85,B 0,C 180,E1 12209.367,E2 12209.367} C_VEL
LIN {X 0,Y 310.269,Z 645.746,A -85,B 0,C 180,E1 12208.467,E2 12208.467} C_VEL
LIN {X 0,Y 305.22,Z 665.866,A -85,B 0,C 180,E1 12207.338,E2 12207.338} C_VEL
LIN {X 0,Y 299.341,Z 685.31,A -85,B 0,C 180,E1 12205.929,E2 12205.929} C_VEL
LIN {X 0,Y 292.719,Z 704.148,A -85,B 0,C 180,E1 12204.215,E2 12204.215} C_VEL
LIN {X 0,Y 285.512,Z 722.428,A -85,B 0,C 180,E1 12202.155,E2 12202.155} C_VEL
LIN {X 0,Y 277.872,Z 739.964,A -85,B 0,C 180,E1 12199.713,E2 12199.713} C_VEL
LIN {X 0,Y 269.992,Z 756.507,A -85,B 0,C 180,E1 12196.847,E2 12196.847} C_VEL
LIN {X 0,Y 262.362,Z 771.703,A -85,B 0,C 180,E1 12193.608,E2 12193.608} C_VEL
LIN {X 0,Y 255.165,Z 785.577,A -85,B 0,C 180,E1 12189.987,E2 12189.987} C_VEL
LIN {X 0,Y 248.633,Z 798.077,A -85,B 0,C 180,E1 12185.952,E2 12185.952} C_VEL
LIN {X 0,Y 242.963,Z 809.17,A -85,B 0,C 180,E1 12181.508,E2 12181.508} C_VEL
LIN {X 0,Y 238.193,Z 819.314,A -85,B 0,C 180,E1 12176.42,E2 12176.42} C_VEL
LIN {X 0,Y 235.047,Z 827.114,A -85,B 0,C 180,E1 12171.458,E2 12171.458} C_VEL
LIN {X 0,Y 233.145,Z 833.119,A -85,B 0,C 180,E1 12166.442,E2 12166.442} C_VEL
LIN {X 0,Y 232.263,Z 837.685,A -85,B 0,C 180,E1 12161.17,E2 12161.17} C_VEL
LIN {X 0,Y 232.114,Z 840.387,A -85,B 0,C 180,E1 12156.43,E2 12156.43} C_VEL
LIN {X 0,Y 232.188,Z 841.533,A -85,B 0,C 180,E1 12151.974,E2 12151.974} C_VEL
LIN {X 0,Y 232.188,Z 841.53,A -85,B 0,C 180,E1 12148.026,E2 12148.026} C_VEL
LIN {X 0,Y 232.118,Z 840.25,A -85,B 0,C 180,E1 12143.321,E2 12143.321} C_VEL
LIN {X 0,Y 232.263,Z 837.666,A -85,B 0,C 180,E1 12138.83,E2 12138.83} C_VEL
LIN {X 0,Y 233.145,Z 833.092,A -85,B 0,C 180,E1 12133.558,E2 12133.558} C_VEL
LIN {X 0,Y 235.046,Z 827.084,A -85,B 0,C 180,E1 12128.542,E2 12128.542} C_VEL
LIN {X 0,Y 238.188,Z 819.268,A -85,B 0,C 180,E1 12123.58,E2 12123.58} C_VEL
LIN {X 0,Y 242.959,Z 809.11,A -85,B 0,C 180,E1 12118.491,E2 12118.491} C_VEL
LIN {X 0,Y 248.628,Z 798.005,A -85,B 0,C 180,E1 12114.047,E2 12114.047} C_VEL
LIN {X 0,Y 255.158,Z 785.494,A -85,B 0,C 180,E1 12110.012,E2 12110.012} C_VEL
LIN {X 0,Y 262.358,Z 771.585,A -85,B 0,C 180,E1 12106.387,E2 12106.387} C_VEL
LIN {X 0,Y 270.482,Z 755.334,A -85,B 0,C 180,E1 12102.954,E2 12102.954} C_VEL
LIN {X 0,Y 278.402,Z 738.556,A -85,B 0,C 180,E1 12100.097,E2 12100.097} C_VEL
LIN {X 0,Y 286.06,Z 720.954,A -85,B 0,C 180,E1 12097.676,E2 12097.676} C_VEL
LIN {X 0,Y 293.317,Z 702.278,A -85,B 0,C 180,E1 12095.612,E2 12095.612} C_VEL
LIN {X 0,Y 299.96,Z 682.995,A -85,B 0,C 180,E1 12093.904,E2 12093.904} C_VEL
LIN {X 0,Y 305.864,Z 663.109,A -85,B 0,C 180,E1 12092.502,E2 12092.502} C_VEL
LIN {X 0,Y 310.934,Z 642.363,A -85,B 0,C 180,E1 12091.38,E2 12091.38} C_VEL
LIN {X 0,Y 315.035,Z 620.894,A -85,B 0,C 180,E1 12090.524,E2 12090.524} C_VEL
LIN {X 0,Y 318.068,Z 597.726,A -85,B 0,C 180,E1 12089.86,E2 12089.86} C_VEL
LIN {X 0,Y 331.661,Z 422.246,A -85,B 0,C 180,E1 12086.089,E2 12086.089} C_VEL
LIN {X 0,Y 324.725,Z 409.766,A -85,B 0,C 180,E1 12083.115,E2 12083.115} C_VEL
LIN {X 0,Y 317.766,Z 398.258,A -85,B 0,C 180,E1 12079.674,E2 12079.674} C_VEL
LIN {X 0,Y 312.118,Z 389.697,A -85,B 0,C 180,E1 12076.374,E2 12076.374} C_VEL
LIN {X 0,Y 308.867,Z 385.017,A -85,B 0,C 180,E1 12074.146,E2 12074.146} C_VEL
LIN {X 0,Y 305.703,Z 380.471,A -85,B 0,C 180,E1 12071.604,E2 12071.604} C_VEL
LIN {X 0,Y 302.308,Z 375.701,A -85,B 0,C 180,E1 12068.176,E2 12068.176} C_VEL
LIN {X 0,Y 298.582,Z 370.641,A -85,B 0,C 180,E1 12061.919,E2 12061.919} C_VEL
LIN {X 0,Y 297.763,Z 370.161,A -85,B 0,C 180,E1 12056.727,E2 12056.727} C_VEL
LIN {X 0,Y 298.303,Z 370.949,A -85,B 0,C 180,E1 12053.649,E2 12053.649} C_VEL
LIN {X 0,Y 301.449,Z 375.989,A -85,B 0,C 180,E1 12047.646,E2 12047.646} C_VEL
LIN {X 0,Y 304.506,Z 380.613,A -85,B 0,C 180,E1 12044.282,E2 12044.282} C_VEL
LIN {X 0,Y 308.066,Z 386.103,A -85,B 0,C 180,E1 12041.257,E2 12041.257} C_VEL
LIN {X 0,Y 312.822,Z 393.584,A -85,B 0,C 180,E1 12037.99,E2 12037.99} C_VEL
LIN {X 0,Y 317.735,Z 401.694,A -85,B 0,C 180,E1 12035.159,E2 12035.159} C_VEL
LIN {X 0,Y 324.143,Z 412.939,A -85,B 0,C 180,E1 12031.989,E2 12031.989} C_VEL
LIN {X 0,Y 330.104,Z 424.349,A -85,B 0,C 180,E1 12029.399,E2 12029.399} C_VEL
LIN {X 0,Y 317.661,Z 597.677,A -85,B 0,C 180,E1 12025.862,E2 12025.862} C_VEL
LIN {X 0,Y 314.691,Z 619.024,A -85,B 0,C 180,E1 12025.201,E2 12025.201} C_VEL
LIN {X 0,Y 310.782,Z 638.975,A -85,B 0,C 180,E1 12024.324,E2 12024.324} C_VEL
LIN {X 0,Y 305.621,Z 659.508,A -85,B 0,C 180,E1 12023.118,E2 12023.118} C_VEL
LIN {X 0,Y 299.979,Z 678.035,A -85,B 0,C 180,E1 12021.713,E2 12021.713} C_VEL
LIN {X 0,Y 293.289,Z 696.556,A -85,B 0,C 180,E1 12019.936,E2 12019.936} C_VEL
LIN {X 0,Y 286.157,Z 713.725,A -85,B 0,C 180,E1 12017.866,E2 12017.866} C_VEL
LIN {X 0,Y 278.594,Z 730.022,A -85,B 0,C 180,E1 12015.429,E2 12015.429} C_VEL
LIN {X 0,Y 271.164,Z 744.68,A -85,B 0,C 180,E1 12012.722,E2 12012.722} C_VEL
LIN {X 0,Y 263.652,Z 758.425,A -85,B 0,C 180,E1 12009.576,E2 12009.576} C_VEL
LIN {X 0,Y 256.503,Z 770.716,A -85,B 0,C 180,E1 12006.057,E2 12006.057} C_VEL
LIN {X 0,Y 249.956,Z 781.676,A -85,B 0,C 180,E1 12002.141,E2 12002.141} C_VEL
LIN {X 0,Y 244.221,Z 791.275,A -85,B 0,C 180,E1 11997.821,E2 11997.821} C_VEL
LIN {X 0,Y 239.502,Z 799.448,A -85,B 0,C 180,E1 11993.105,E2 11993.105} C_VEL
LIN {X 0,Y 235.969,Z 806.022,A -85,B 0,C 180,E1 11988.018,E2 11988.018} C_VEL
LIN {X 0,Y 233.848,Z 810.591,A -85,B 0,C 180,E1 11983.097,E2 11983.097} C_VEL
LIN {X 0,Y 232.708,Z 813.787,A -85,B 0,C 180,E1 11977.903,E2 11977.903} C_VEL
LIN {X 0,Y 232.321,Z 815.394,A -85,B 0,C 180,E1 11972.96,E2 11972.96} C_VEL
LIN {X 0,Y 232.282,Z 815.517,A -85,B 0,C 180,E1 11968.273,E2 11968.273} C_VEL
LIN {X 0,Y 232.553,Z 814.36,A -85,B 0,C 180,E1 11963.309,E2 11963.309} C_VEL
LIN {X 0,Y 233.41,Z 811.798,A -85,B 0,C 180,E1 11958.385,E2 11958.385} C_VEL
LIN {X 0,Y 235.165,Z 807.659,A -85,B 0,C 180,E1 11953.45,E2 11953.45} C_VEL
LIN {X 0,Y 238.286,Z 801.627,A -85,B 0,C 180,E1 11948.331,E2 11948.331} C_VEL
LIN {X 0,Y 242.587,Z 794.122,A -85,B 0,C 180,E1 11943.569,E2 11943.569} C_VEL
LIN {X 0,Y 248.238,Z 784.696,A -85,B 0,C 180,E1 11938.966,E2 11938.966} C_VEL
LIN {X 0,Y 254.857,Z 773.66,A -85,B 0,C 180,E1 11934.782,E2 11934.782} C_VEL
LIN {X 0,Y 261.858,Z 761.634,A -85,B 0,C 180,E1 11931.164,E2 11931.164} C_VEL
LIN {X 0,Y 269.564,Z 747.798,A -85,B 0,C 180,E1 11927.829,E2 11927.829} C_VEL
LIN {X 0,Y 277.132,Z 733.229,A -85,B 0,C 180,E1 11924.999,E2 11924.999} C_VEL
LIN {X 0,Y 284.746,Z 717.226,A -85,B 0,C 180,E1 11922.492,E2 11922.492} C_VEL
LIN {X 0,Y 292.132,Z 699.733,A -85,B 0,C 180,E1 11920.307,E2 11920.307} C_VEL
LIN {X 0,Y 298.583,Z 682.368,A -85,B 0,C 180,E1 11918.566,E2 11918.566} C_VEL
LIN {X 0,Y 304.52,Z 663.852,A -85,B 0,C 180,E1 11917.075,E2 11917.075} C_VEL
LIN {X 0,Y 309.66,Z 644.61,A -85,B 0,C 180,E1 11915.862,E2 11915.862} C_VEL
LIN {X 0,Y 313.947,Z 623.992,A -85,B 0,C 180,E1 11914.888,E2 11914.888} C_VEL
LIN {X 0,Y 317.112,Z 603.122,A -85,B 0,C 180,E1 11914.183,E2 11914.183} C_VEL
LIN {X 0,Y 319.542,Z 575.466,A -85,B 0,C 180,E1 11913.553,E2 11913.553} C_VEL
LIN {X 0,Y 324.493,Z 504.139,A -85,B 0,C 180,E1 11912.099,E2 11912.099} C_VEL
LIN {X 0,Y 324.533,Z 496.57,A -85,B 0,C 180,E1 11911.792,E2 11911.792} C_VEL
LIN {X 0,Y 322.952,Z 476.843,A -85,B 0,C 180,E1 11910.424,E2 11910.424} C_VEL
LIN {X 0,Y 323.075,Z 470.336,A -85,B 0,C 180,E1 11910.173,E2 11910.173} C_VEL
LIN {X 0,Y 326.185,Z 428.443,A -85,B 0,C 180,E1 11909.32,E2 11909.32} C_VEL
LIN {X 0,Y 319.931,Z 416.407,A -85,B 0,C 180,E1 11906.396,E2 11906.396} C_VEL
LIN {X 0,Y 314.247,Z 406.321,A -85,B 0,C 180,E1 11903.337,E2 11903.337} C_VEL
LIN {X 0,Y 309.356,Z 398.184,A -85,B 0,C 180,E1 11900.233,E2 11900.233} C_VEL
LIN {X 0,Y 305.342,Z 391.727,A -85,B 0,C 180,E1 11897.14,E2 11897.14} C_VEL
LIN {X 0,Y 302.344,Z 386.97,A -85,B 0,C 180,E1 11894.263,E2 11894.263} C_VEL
LIN {X 0,Y 299.869,Z 383.082,A -85,B 0,C 180,E1 11891.151,E2 11891.151} C_VEL
LIN {X 0,Y 297.282,Z 378.538,A -85,B 0,C 180,E1 11885.017,E2 11885.017} C_VEL
LIN {X 0,Y 297.371,Z 378.404,A -85,B 0,C 180,E1 11879.615,E2 11879.615} C_VEL
LIN {X 0,Y 298.085,Z 379.422,A -85,B 0,C 180,E1 11877.309,E2 11877.309} C_VEL
LIN {X 0,Y 301.674,Z 384.264,A -85,B 0,C 180,E1 11871.615,E2 11871.615} C_VEL
LIN {X 0,Y 305.299,Z 389.569,A -85,B 0,C 180,E1 11867.997,E2 11867.997} C_VEL
LIN {X 0,Y 308.951,Z 394.994,A -85,B 0,C 180,E1 11865.139,E2 11865.139} C_VEL
LIN {X 0,Y 313.593,Z 402.006,A -85,B 0,C 180,E1 11862.129,E2 11862.129} C_VEL
LIN {X 0,Y 320.036,Z 412.704,A -85,B 0,C 180,E1 11858.608,E2 11858.608} C_VEL
LIN {X 0,Y 326.597,Z 424.465,A -85,B 0,C 180,E1 11855.54,E2 11855.54} C_VEL
LIN {X 0,Y 327.69,Z 426.847,A -85,B 0,C 180,E1 11855.05,E2 11855.05} C_VEL
LIN {X 0,Y 313.557,Z 602.443,A -85,B 0,C 180,E1 11851.281,E2 11851.281} C_VEL
LIN {X 0,Y 310.289,Z 624.385,A -85,B 0,C 180,E1 11850.612,E2 11850.612} C_VEL
LIN {X 0,Y 305.919,Z 645.504,A -85,B 0,C 180,E1 11849.728,E2 11849.728} C_VEL
LIN {X 0,Y 300.554,Z 666.205,A -85,B 0,C 180,E1 11848.57,E2 11848.57} C_VEL
LIN {X 0,Y 294.506,Z 685.585,A -85,B 0,C 180,E1 11847.166,E2 11847.166} C_VEL
LIN {X 0,Y 287.679,Z 704.321,A -85,B 0,C 180,E1 11845.456,E2 11845.456} C_VEL
LIN {X 0,Y 279.93,Z 723.202,A -85,B 0,C 180,E1 11843.307,E2 11843.307} C_VEL
LIN {X 0,Y 272.034,Z 740.596,A -85,B 0,C 180,E1 11840.851,E2 11840.851} C_VEL
LIN {X 0,Y 263.869,Z 757.009,A -85,B 0,C 180,E1 11837.959,E2 11837.959} C_VEL
LIN {X 0,Y 255.94,Z 772.049,A -85,B 0,C 180,E1 11834.682,E2 11834.682} C_VEL
LIN {X 0,Y 248.426,Z 785.808,A -85,B 0,C 180,E1 11830.997,E2 11830.997} C_VEL
LIN {X 0,Y 241.587,Z 798.245,A -85,B 0,C 180,E1 11826.877,E2 11826.877} C_VEL
LIN {X 0,Y 235.621,Z 809.226,A -85,B 0,C 180,E1 11822.321,E2 11822.321} C_VEL
LIN {X 0,Y 230.78,Z 818.841,A -85,B 0,C 180,E1 11817.338,E2 11817.338} C_VEL
LIN {X 0,Y 227.375,Z 826.648,A -85,B 0,C 180,E1 11812.22,E2 11812.22} C_VEL
LIN {X 0,Y 225.29,Z 832.656,A -85,B 0,C 180,E1 11807.032,E2 11807.032} C_VEL
LIN {X 0,Y 224.297,Z 837.229,A -85,B 0,C 180,E1 11801.572,E2 11801.572} C_VEL
LIN {X 0,Y 224.126,Z 839.935,A -85,B 0,C 180,E1 11796.661,E2 11796.661} C_VEL
LIN {X 0,Y 224.199,Z 841.085,A -85,B 0,C 180,E1 11792.045,E2 11792.045} C_VEL
LIN {X 0,Y 224.202,Z 841.107,A -85,B 0,C 180,E1 11788.211,E2 11788.211} C_VEL
LIN {X 0,Y 224.122,Z 840.03,A -85,B 0,C 180,E1 11783.597,E2 11783.597} C_VEL
LIN {X 0,Y 224.276,Z 837.381,A -85,B 0,C 180,E1 11778.688,E2 11778.688} C_VEL
LIN {X 0,Y 225.146,Z 833.171,A -85,B 0,C 180,E1 11773.488,E2 11773.488} C_VEL
LIN {X 0,Y 227.13,Z 827.211,A -85,B 0,C 180,E1 11768.255,E2 11768.255} C_VEL
LIN {X 0,Y 230.576,Z 819.22,A -85,B 0,C 180,E1 11762.915,E2 11762.915} C_VEL
LIN {X 0,Y 235.341,Z 809.704,A -85,B 0,C 180,E1 11757.923,E2 11757.923} C_VEL
LIN {X 0,Y 241.235,Z 798.813,A -85,B 0,C 180,E1 11753.357,E2 11753.357} C_VEL
LIN {X 0,Y 248.005,Z 786.448,A -85,B 0,C 180,E1 11749.224,E2 11749.224} C_VEL
LIN {X 0,Y 255.463,Z 772.813,A -85,B 0,C 180,E1 11745.527,E2 11745.527} C_VEL
LIN {X 0,Y 263.413,Z 757.772,A -85,B 0,C 180,E1 11742.21,E2 11742.21} C_VEL
LIN {X 0,Y 271.589,Z 741.31,A -85,B 0,C 180,E1 11739.288,E2 11739.288} C_VEL
LIN {X 0,Y 279.307,Z 724.379,A -85,B 0,C 180,E1 11736.864,E2 11736.864} C_VEL
LIN {X 0,Y 287.345,Z 704.919,A -85,B 0,C 180,E1 11734.623,E2 11734.623} C_VEL
LIN {X 0,Y 294.161,Z 686.317,A -85,B 0,C 180,E1 11732.909,E2 11732.909} C_VEL
LIN {X 0,Y 300.537,Z 665.872,A -85,B 0,C 180,E1 11731.425,E2 11731.425} C_VEL
LIN {X 0,Y 305.902,Z 645.077,A -85,B 0,C 180,E1 11730.266,E2 11730.266} C_VEL
LIN {X 0,Y 310.49,Z 622.482,A -85,B 0,C 180,E1 11729.336,E2 11729.336} C_VEL
LIN {X 0,Y 313.617,Z 600.475,A -85,B 0,C 180,E1 11728.686,E2 11728.686} C_VEL
LIN {X 0,Y 327.547,Z 426.402,A -85,B 0,C 180,E1 11724.938,E2 11724.938} C_VEL
LIN {X 0,Y 321.512,Z 415.449,A -85,B 0,C 180,E1 11722.2,E2 11722.2} C_VEL
LIN {X 0,Y 315.46,Z 405.143,A -85,B 0,C 180,E1 11719.054,E2 11719.054} C_VEL
LIN {X 0,Y 310.007,Z 396.674,A -85,B 0,C 180,E1 11715.719,E2 11715.719} C_VEL
LIN {X 0,Y 307.004,Z 392.242,A -85,B 0,C 180,E1 11713.561,E2 11713.561} C_VEL
LIN {X 0,Y 304.178,Z 388.041,A -85,B 0,C 180,E1 11711.182,E2 11711.182} C_VEL
LIN {X 0,Y 300.993,Z 383.43,A -85,B 0,C 180,E1 11707.827,E2 11707.827} C_VEL
LIN {X 0,Y 297.533,Z 378.537,A -85,B 0,C 180,E1 11701.733,E2 11701.733} C_VEL
LIN {X 0,Y 296.79,Z 378.105,A -85,B 0,C 180,E1 11696.716,E2 11696.716} C_VEL
LIN {X 0,Y 297.275,Z 378.834,A -85,B 0,C 180,E1 11693.821,E2 11693.821} C_VEL
LIN {X 0,Y 300.194,Z 383.692,A -85,B 0,C 180,E1 11687.985,E2 11687.985} C_VEL
LIN {X 0,Y 303.149,Z 388.354,A -85,B 0,C 180,E1 11684.602,E2 11684.602} C_VEL
LIN {X 0,Y 306.502,Z 393.685,A -85,B 0,C 180,E1 11681.651,E2 11681.651} C_VEL
LIN {X 0,Y 310.999,Z 400.992,A -85,B 0,C 180,E1 11678.45,E2 11678.45} C_VEL
LIN {X 0,Y 315.631,Z 408.871,A -85,B 0,C 180,E1 11675.681,E2 11675.681} C_VEL
LIN {X 0,Y 321.795,Z 420.013,A -85,B 0,C 180,E1 11672.522,E2 11672.522} C_VEL
LIN {X 0,Y 326.073,Z 428.633,A -85,B 0,C 180,E1 11670.554,E2 11670.554} C_VEL
LIN {X 0,Y 313.479,Z 597.862,A -85,B 0,C 180,E1 11667.101,E2 11667.101} C_VEL
LIN {X 0,Y 310.401,Z 619.334,A -85,B 0,C 180,E1 11666.439,E2 11666.439} C_VEL
LIN {X 0,Y 306.386,Z 639.224,A -85,B 0,C 180,E1 11665.568,E2 11665.568} C_VEL
LIN {X 0,Y 301.238,Z 659.183,A -85,B 0,C 180,E1 11664.407,E2 11664.407} C_VEL
LIN {X 0,Y 295.422,Z 677.826,A -85,B 0,C 180,E1 11663.008,E2 11663.008} C_VEL
LIN {X 0,Y 288.51,Z 696.399,A -85,B 0,C 180,E1 11661.236,E2 11661.236} C_VEL
LIN {X 0,Y 281.284,Z 713.311,A -85,B 0,C 180,E1 11659.21,E2 11659.21} C_VEL
LIN {X 0,Y 273.084,Z 730.419,A -85,B 0,C 180,E1 11656.655,E2 11656.655} C_VEL
LIN {X 0,Y 265.297,Z 745.187,A -85,B 0,C 180,E1 11653.903,E2 11653.903} C_VEL
LIN {X 0,Y 257.477,Z 758.925,A -85,B 0,C 180,E1 11650.721,E2 11650.721} C_VEL
LIN {X 0,Y 250.004,Z 771.201,A -85,B 0,C 180,E1 11647.149,E2 11647.149} C_VEL
LIN {X 0,Y 243.131,Z 782.149,A -85,B 0,C 180,E1 11643.157,E2 11643.157} C_VEL
LIN {X 0,Y 236.957,Z 791.923,A -85,B 0,C 180,E1 11638.636,E2 11638.636} C_VEL
LIN {X 0,Y 232.067,Z 799.908,A -85,B 0,C 180,E1 11633.89,E2 11633.89} C_VEL
LIN {X 0,Y 228.288,Z 806.48,A -85,B 0,C 180,E1 11628.646,E2 11628.646} C_VEL
LIN {X 0,Y 226.002,Z 811.045,A -85,B 0,C 180,E1 11623.56,E2 11623.56} C_VEL
LIN {X 0,Y 224.761,Z 814.238,A -85,B 0,C 180,E1 11618.184,E2 11618.184} C_VEL
LIN {X 0,Y 224.337,Z 815.843,A -85,B 0,C 180,E1 11613.066,E2 11613.066} C_VEL
LIN {X 0,Y 224.296,Z 815.965,A -85,B 0,C 180,E1 11608.212,E2 11608.212} C_VEL
LIN {X 0,Y 224.59,Z 814.821,A -85,B 0,C 180,E1 11603.096,E2 11603.096} C_VEL
LIN {X 0,Y 225.525,Z 812.249,A -85,B 0,C 180,E1 11597.973,E2 11597.973} C_VEL
LIN {X 0,Y 227.557,Z 807.873,A -85,B 0,C 180,E1 11592.616,E2 11592.616} C_VEL
LIN {X 0,Y 230.966,Z 801.75,A -85,B 0,C 180,E1 11587.339,E2 11587.339} C_VEL
LIN {X 0,Y 235.614,Z 794.146,A -85,B 0,C 180,E1 11582.449,E2 11582.449} C_VEL
LIN {X 0,Y 241.323,Z 785.166,A -85,B 0,C 180,E1 11577.973,E2 11577.973} C_VEL
LIN {X 0,Y 248.282,Z 774.132,A -85,B 0,C 180,E1 11573.703,E2 11573.703} C_VEL
LIN {X 0,Y 255.502,Z 762.297,A -85,B 0,C 180,E1 11570.077,E2 11570.077} C_VEL
LIN {X 0,Y 263.639,Z 748.302,A -85,B 0,C 180,E1 11566.652,E2 11566.652} C_VEL
LIN {X 0,Y 271.501,Z 733.76,A -85,B 0,C 180,E1 11563.797,E2 11563.797} C_VEL
LIN {X 0,Y 279.388,Z 717.775,A -85,B 0,C 180,E1 11561.278,E2 11561.278} C_VEL
LIN {X 0,Y 286.519,Z 701.507,A -85,B 0,C 180,E1 11559.223,E2 11559.223} C_VEL
LIN {X 0,Y 293.671,Z 683.037,A -85,B 0,C 180,E1 11557.347,E2 11557.347} C_VEL
LIN {X 0,Y 299.785,Z 664.633,A -85,B 0,C 180,E1 11555.861,E2 11555.861} C_VEL
LIN {X 0,Y 305.069,Z 645.471,A -85,B 0,C 180,E1 11554.652,E2 11554.652} C_VEL
LIN {X 0,Y 309.463,Z 625.168,A -85,B 0,C 180,E1 11553.686,E2 11553.686} C_VEL
LIN {X 0,Y 312.838,Z 603.908,A -85,B 0,C 180,E1 11552.96,E2 11552.96} C_VEL
LIN {X 0,Y 315.178,Z 579.149,A -85,B 0,C 180,E1 11552.385,E2 11552.385} C_VEL
LIN {X 0,Y 323.075,Z 470.336,A -85,B 0,C 180,E1 11550.173,E2 11550.173} C_VEL
LIN {X 0,Y 323.172,Z 462.769,A -85,B 0,C 180,E1 11549.863,E2 11549.863} C_VEL
LIN {X 0,Y 321.867,Z 443.044,A -85,B 0,C 180,E1 11548.478,E2 11548.478} C_VEL
LIN {X 0,Y 322.049,Z 436.537,A -85,B 0,C 180,E1 11548.23,E2 11548.23} C_VEL
LIN {X 0,Y 322.31,Z 432.607,A -85,B 0,C 180,E1 11548.134,E2 11548.134} C_VEL
LIN {X 0,Y 316.764,Z 421.791,A -85,B 0,C 180,E1 11545.372,E2 11545.372} C_VEL
LIN {X 0,Y 311.153,Z 411.543,A -85,B 0,C 180,E1 11542.134,E2 11542.134} C_VEL
LIN {X 0,Y 306.521,Z 403.663,A -85,B 0,C 180,E1 11538.939,E2 11538.939} C_VEL
LIN {X 0,Y 303.624,Z 398.998,A -85,B 0,C 180,E1 11536.55,E2 11536.55} C_VEL
LIN {X 0,Y 301.031,Z 394.674,A -85,B 0,C 180,E1 11533.934,E2 11533.934} C_VEL
LIN {X 0,Y 298.646,Z 390.832,A -85,B 0,C 180,E1 11530.806,E2 11530.806} C_VEL
LIN {X 0,Y 296.275,Z 386.444,A -85,B 0,C 180,E1 11524.84,E2 11524.84} C_VEL
LIN {X 0,Y 296.396,Z 386.35,A -85,B 0,C 180,E1 11519.614,E2 11519.614} C_VEL
LIN {X 0,Y 297.03,Z 387.299,A -85,B 0,C 180,E1 11517.492,E2 11517.492} C_VEL
LIN {X 0,Y 300.43,Z 392.096,A -85,B 0,C 180,E1 11511.869,E2 11511.869} C_VEL
LIN {X 0,Y 303.861,Z 397.28,A -85,B 0,C 180,E1 11508.325,E2 11508.325} C_VEL
LIN {X 0,Y 307.359,Z 402.635,A -85,B 0,C 180,E1 11505.494,E2 11505.494} C_VEL
LIN {X 0,Y 311.685,Z 409.374,A -85,B 0,C 180,E1 11502.595,E2 11502.595} C_VEL
LIN {X 0,Y 317.8,Z 419.827,A -85,B 0,C 180,E1 11499.127,E2 11499.127} C_VEL
LIN {X 0,Y 323.735,Z 430.828,A -85,B 0,C 180,E1 11496.231,E2 11496.231} C_VEL
LIN {X 0,Y 309.533,Z 602.281,A -85,B 0,C 180,E1 11492.558,E2 11492.558} C_VEL
LIN {X 0,Y 306.184,Z 624.245,A -85,B 0,C 180,E1 11491.895,E2 11491.895} C_VEL
LIN {X 0,Y 301.72,Z 645.266,A -85,B 0,C 180,E1 11491.025,E2 11491.025} C_VEL
LIN {X 0,Y 296.263,Z 665.797,A -85,B 0,C 180,E1 11489.89,E2 11489.89} C_VEL
LIN {X 0,Y 289.813,Z 685.864,A -85,B 0,C 180,E1 11488.444,E2 11488.444} C_VEL
LIN {X 0,Y 282.811,Z 704.412,A -85,B 0,C 180,E1 11486.75,E2 11486.75} C_VEL
LIN {X 0,Y 274.778,Z 723.292,A -85,B 0,C 180,E1 11484.594,E2 11484.594} C_VEL
LIN {X 0,Y 266.6,Z 740.615,A -85,B 0,C 180,E1 11482.133,E2 11482.133} C_VEL
LIN {X 0,Y 257.851,Z 757.515,A -85,B 0,C 180,E1 11479.123,E2 11479.123} C_VEL
LIN {X 0,Y 249.605,Z 772.408,A -85,B 0,C 180,E1 11475.808,E2 11475.808} C_VEL
LIN {X 0,Y 241.337,Z 786.765,A -85,B 0,C 180,E1 11471.836,E2 11471.836} C_VEL
LIN {X 0,Y 234.24,Z 798.997,A -85,B 0,C 180,E1 11467.617,E2 11467.617} C_VEL
LIN {X 0,Y 227.752,Z 810.363,A -85,B 0,C 180,E1 11462.681,E2 11462.681} C_VEL
LIN {X 0,Y 222.786,Z 819.65,A -85,B 0,C 180,E1 11457.532,E2 11457.532} C_VEL
LIN {X 0,Y 219.178,Z 827.476,A -85,B 0,C 180,E1 11451.966,E2 11451.966} C_VEL
LIN {X 0,Y 217.148,Z 833.245,A -85,B 0,C 180,E1 11446.587,E2 11446.587} C_VEL
LIN {X 0,Y 216.267,Z 837.293,A -85,B 0,C 180,E1 11441.196,E2 11441.196} C_VEL
LIN {X 0,Y 216.141,Z 839.819,A -85,B 0,C 180,E1 11435.841,E2 11435.841} C_VEL
LIN {X 0,Y 216.217,Z 840.687,A -85,B 0,C 180,E1 11431.59,E2 11431.59} C_VEL
LIN {X 0,Y 216.199,Z 840.581,A -85,B 0,C 180,E1 11427.349,E2 11427.349} C_VEL
LIN {X 0,Y 216.133,Z 839.221,A -85,B 0,C 180,E1 11422.558,E2 11422.558} C_VEL
LIN {X 0,Y 216.366,Z 836.576,A -85,B 0,C 180,E1 11417.727,E2 11417.727} C_VEL
LIN {X 0,Y 217.537,Z 831.89,A -85,B 0,C 180,E1 11412.065,E2 11412.065} C_VEL
LIN {X 0,Y 219.89,Z 825.816,A -85,B 0,C 180,E1 11406.698,E2 11406.698} C_VEL
LIN {X 0,Y 223.648,Z 817.887,A -85,B 0,C 180,E1 11401.422,E2 11401.422} C_VEL
LIN {X 0,Y 228.915,Z 808.139,A -85,B 0,C 180,E1 11396.31,E2 11396.31} C_VEL
LIN {X 0,Y 235.333,Z 797.011,A -85,B 0,C 180,E1 11391.662,E2 11391.662} C_VEL
LIN {X 0,Y 242.639,Z 784.492,A -85,B 0,C 180,E1 11387.485,E2 11387.485} C_VEL
LIN {X 0,Y 250.574,Z 770.546,A -85,B 0,C 180,E1 11383.762,E2 11383.762} C_VEL
LIN {X 0,Y 259.086,Z 754.987,A -85,B 0,C 180,E1 11380.416,E2 11380.416} C_VEL
LIN {X 0,Y 267.467,Z 738.644,A -85,B 0,C 180,E1 11377.581,E2 11377.581} C_VEL
LIN {X 0,Y 275.707,Z 721.051,A -85,B 0,C 180,E1 11375.139,E2 11375.139} C_VEL
LIN {X 0,Y 283.416,Z 702.606,A -85,B 0,C 180,E1 11373.086,E2 11373.086} C_VEL
LIN {X 0,Y 290.811,Z 682.506,A -85,B 0,C 180,E1 11371.31,E2 11371.31} C_VEL
LIN {X 0,Y 297.067,Z 662.611,A -85,B 0,C 180,E1 11369.927,E2 11369.927} C_VEL
LIN {X 0,Y 302.606,Z 641.101,A -85,B 0,C 180,E1 11368.788,E2 11368.788} C_VEL
LIN {X 0,Y 306.873,Z 619.584,A -85,B 0,C 180,E1 11367.962,E2 11367.962} C_VEL
LIN {X 0,Y 309.921,Z 596.99,A -85,B 0,C 180,E1 11367.329,E2 11367.329} C_VEL
LIN {X 0,Y 323.604,Z 430.737,A -85,B 0,C 180,E1 11363.779,E2 11363.779} C_VEL
LIN {X 0,Y 317.403,Z 419.305,A -85,B 0,C 180,E1 11360.756,E2 11360.756} C_VEL
LIN {X 0,Y 311.378,Z 408.999,A -85,B 0,C 180,E1 11357.327,E2 11357.327} C_VEL
LIN {X 0,Y 306.244,Z 400.815,A -85,B 0,C 180,E1 11353.788,E2 11353.788} C_VEL
LIN {X 0,Y 302.67,Z 395.608,A -85,B 0,C 180,E1 11350.757,E2 11350.757} C_VEL
LIN {X 0,Y 299.69,Z 391.157,A -85,B 0,C 180,E1 11347.476,E2 11347.476} C_VEL
LIN {X 0,Y 296.485,Z 386.435,A -85,B 0,C 180,E1 11341.546,E2 11341.546} C_VEL
LIN {X 0,Y 295.828,Z 386.072,A -85,B 0,C 180,E1 11336.512,E2 11336.512} C_VEL
LIN {X 0,Y 296.296,Z 386.855,A -85,B 0,C 180,E1 11333.8,E2 11333.8} C_VEL
LIN {X 0,Y 299.014,Z 391.536,A -85,B 0,C 180,E1 11328.23,E2 11328.23} C_VEL
LIN {X 0,Y 301.798,Z 396.091,A -85,B 0,C 180,E1 11324.925,E2 11324.925} C_VEL
LIN {X 0,Y 304.953,Z 401.263,A -85,B 0,C 180,E1 11322.049,E2 11322.049} C_VEL
LIN {X 0,Y 309.263,Z 408.521,A -85,B 0,C 180,E1 11318.87,E2 11318.87} C_VEL
LIN {X 0,Y 313.627,Z 416.17,A -85,B 0,C 180,E1 11316.171,E2 11316.171} C_VEL
LIN {X 0,Y 319.472,Z 427.106,A -85,B 0,C 180,E1 11313.062,E2 11313.062} C_VEL
LIN {X 0,Y 322.182,Z 432.894,A -85,B 0,C 180,E1 11311.739,E2 11311.739} C_VEL
LIN {X 0,Y 309.468,Z 597.853,A -85,B 0,C 180,E1 11308.377,E2 11308.377} C_VEL
LIN {X 0,Y 306.32,Z 619.281,A -85,B 0,C 180,E1 11307.723,E2 11307.723} C_VEL
LIN {X 0,Y 302.138,Z 639.469,A -85,B 0,C 180,E1 11306.848,E2 11306.848} C_VEL
LIN {X 0,Y 296.675,Z 659.977,A -85,B 0,C 180,E1 11305.657,E2 11305.657} C_VEL
LIN {X 0,Y 290.69,Z 678.503,A -85,B 0,C 180,E1 11304.265,E2 11304.265} C_VEL
LIN {X 0,Y 283.572,Z 697.036,A -85,B 0,C 180,E1 11302.496,E2 11302.496} C_VEL
LIN {X 0,Y 276.113,Z 713.889,A -85,B 0,C 180,E1 11300.47,E2 11300.47} C_VEL
LIN {X 0,Y 267.843,Z 730.554,A -85,B 0,C 180,E1 11297.975,E2 11297.975} C_VEL
LIN {X 0,Y 259.549,Z 745.694,A -85,B 0,C 180,E1 11295.137,E2 11295.137} C_VEL
LIN {X 0,Y 251.41,Z 759.425,A -85,B 0,C 180,E1 11291.922,E2 11291.922} C_VEL
LIN {X 0,Y 243.6,Z 771.683,A -85,B 0,C 180,E1 11288.299,E2 11288.299} C_VEL
LIN {X 0,Y 236.388,Z 782.62,A -85,B 0,C 180,E1 11284.231,E2 11284.231} C_VEL
LIN {X 0,Y 229.996,Z 792.204,A -85,B 0,C 180,E1 11279.708,E2 11279.708} C_VEL
LIN {X 0,Y 224.678,Z 800.367,A -85,B 0,C 180,E1 11274.728,E2 11274.728} C_VEL
LIN {X 0,Y 220.636,Z 806.939,A -85,B 0,C 180,E1 11269.318,E2 11269.318} C_VEL
LIN {X 0,Y 218.168,Z 811.499,A -85,B 0,C 180,E1 11264.057,E2 11264.057} C_VEL
LIN {X 0,Y 216.818,Z 814.689,A -85,B 0,C 180,E1 11258.486,E2 11258.486} C_VEL
LIN {X 0,Y 216.362,Z 816.232,A -85,B 0,C 180,E1 11253.444,E2 11253.444} C_VEL
LIN {X 0,Y 216.305,Z 816.434,A -85,B 0,C 180,E1 11248.411,E2 11248.411} C_VEL
LIN {X 0,Y 216.576,Z 815.483,A -85,B 0,C 180,E1 11243.373,E2 11243.373} C_VEL
LIN {X 0,Y 217.506,Z 812.998,A -85,B 0,C 180,E1 11238.062,E2 11238.062} C_VEL
LIN {X 0,Y 219.579,Z 808.807,A -85,B 0,C 180,E1 11232.511,E2 11232.511} C_VEL
LIN {X 0,Y 223.093,Z 802.88,A -85,B 0,C 180,E1 11227.051,E2 11227.051} C_VEL
LIN {X 0,Y 227.895,Z 795.488,A -85,B 0,C 180,E1 11222.002,E2 11222.002} C_VEL
LIN {X 0,Y 234.134,Z 786.142,A -85,B 0,C 180,E1 11217.158,E2 11217.158} C_VEL
LIN {X 0,Y 240.969,Z 775.832,A -85,B 0,C 180,E1 11213.013,E2 11213.013} C_VEL
LIN {X 0,Y 248.884,Z 763.53,A -85,B 0,C 180,E1 11209.095,E2 11209.095} C_VEL
LIN {X 0,Y 257.312,Z 749.708,A -85,B 0,C 180,E1 11205.619,E2 11205.619} C_VEL
LIN {X 0,Y 265.752,Z 734.764,A -85,B 0,C 180,E1 11202.628,E2 11202.628} C_VEL
LIN {X 0,Y 274.158,Z 718.321,A -85,B 0,C 180,E1 11200.017,E2 11200.017} C_VEL
LIN {X 0,Y 282.005,Z 701.001,A -85,B 0,C 180,E1 11197.835,E2 11197.835} C_VEL
LIN {X 0,Y 289.222,Z 682.815,A -85,B 0,C 180,E1 11196.009,E2 11196.009} C_VEL
LIN {X 0,Y 295.612,Z 663.979,A -85,B 0,C 180,E1 11194.508,E2 11194.508} C_VEL
LIN {X 0,Y 301.134,Z 644.382,A -85,B 0,C 180,E1 11193.294,E2 11193.294} C_VEL
LIN {X 0,Y 305.733,Z 623.296,A -85,B 0,C 180,E1 11192.322,E2 11192.322} C_VEL
LIN {X 0,Y 308.999,Z 602.523,A -85,B 0,C 180,E1 11191.644,E2 11191.644} C_VEL
LIN {X 0,Y 311.562,Z 574.519,A -85,B 0,C 180,E1 11191.016,E2 11191.016} C_VEL
LIN {X 0,Y 322.049,Z 436.537,A -85,B 0,C 180,E1 11188.23,E2 11188.23} C_VEL
LIN {X 0,Y 321.868,Z 433.314,A -85,B 0,C 180,E1 11188.005,E2 11188.005} C_VEL
LIN {X 0,Y 320.785,Z 430.165,A -85,B 0,C 180,E1 11187.44,E2 11187.44} C_VEL
LIN {X 0,Y 318.571,Z 427.458,A -85,B 0,C 180,E1 11186.431,E2 11186.431} C_VEL
LIN {X 0,Y 312.301,Z 423.801,A -85,B 0,C 180,E1 11183.481,E2 11183.481} C_VEL
LIN {X 0,Y 310.865,Z 421.791,A -85,B 0,C 180,E1 11182.654,E2 11182.654} C_VEL
LIN {X 0,Y 305.77,Z 412.731,A -85,B 0,C 180,E1 11179.186,E2 11179.186} C_VEL
LIN {X 0,Y 302.244,Z 406.703,A -85,B 0,C 180,E1 11176.233,E2 11176.233} C_VEL
LIN {X 0,Y 299.645,Z 402.27,A -85,B 0,C 180,E1 11173.508,E2 11173.508} C_VEL
LIN {X 0,Y 297.436,Z 398.58,A -85,B 0,C 180,E1 11170.459,E2 11170.459} C_VEL
LIN {X 0,Y 295.269,Z 394.353,A -85,B 0,C 180,E1 11164.662,E2 11164.662} C_VEL
LIN {X 0,Y 295.42,Z 394.296,A -85,B 0,C 180,E1 11159.613,E2 11159.613} C_VEL
LIN {X 0,Y 295.979,Z 395.176,A -85,B 0,C 180,E1 11157.677,E2 11157.677} C_VEL
LIN {X 0,Y 299.122,Z 399.777,A -85,B 0,C 180,E1 11152.22,E2 11152.22} C_VEL
LIN {X 0,Y 302.336,Z 404.81,A -85,B 0,C 180,E1 11148.749,E2 11148.749} C_VEL
LIN {X 0,Y 305.728,Z 410.176,A -85,B 0,C 180,E1 11145.899,E2 11145.899} C_VEL
LIN {X 0,Y 309.862,Z 416.862,A -85,B 0,C 180,E1 11143.021,E2 11143.021} C_VEL
LIN {X 0,Y 315.504,Z 426.837,A -85,B 0,C 180,E1 11139.696,E2 11139.696} C_VEL
LIN {X 0,Y 319.905,Z 435.392,A -85,B 0,C 180,E1 11137.42,E2 11137.42} C_VEL
LIN {X 0,Y 305.655,Z 602.226,A -85,B 0,C 180,E1 11133.866,E2 11133.866} C_VEL
LIN {X 0,Y 302.211,Z 624.237,A -85,B 0,C 180,E1 11133.207,E2 11133.207} C_VEL
LIN {X 0,Y 297.498,Z 645.776,A -85,B 0,C 180,E1 11132.322,E2 11132.322} C_VEL
LIN {X 0,Y 291.66,Z 666.892,A -85,B 0,C 180,E1 11131.148,E2 11131.148} C_VEL
LIN {X 0,Y 284.922,Z 687.123,A -85,B 0,C 180,E1 11129.683,E2 11129.683} C_VEL
LIN {X 0,Y 277.355,Z 706.324,A -85,B 0,C 180,E1 11127.903,E2 11127.903} C_VEL
LIN {X 0,Y 269.196,Z 724.6,A -85,B 0,C 180,E1 11125.772,E2 11125.772} C_VEL
LIN {X 0,Y 260.501,Z 742.138,A -85,B 0,C 180,E1 11123.219,E2 11123.219} C_VEL
LIN {X 0,Y 251.626,Z 758.584,A -85,B 0,C 180,E1 11120.227,E2 11120.227} C_VEL
LIN {X 0,Y 242.868,Z 773.641,A -85,B 0,C 180,E1 11116.775,E2 11116.775} C_VEL
LIN {X 0,Y 234.509,Z 787.388,A -85,B 0,C 180,E1 11112.833,E2 11112.833} C_VEL
LIN {X 0,Y 226.555,Z 800.308,A -85,B 0,C 180,E1 11108.159,E2 11108.159} C_VEL
LIN {X 0,Y 220.179,Z 810.908,A -85,B 0,C 180,E1 11103.326,E2 11103.326} C_VEL
LIN {X 0,Y 214.895,Z 820.259,A -85,B 0,C 180,E1 11097.869,E2 11097.869} C_VEL
LIN {X 0,Y 211.251,Z 827.655,A -85,B 0,C 180,E1 11092.249,E2 11092.249} C_VEL
LIN {X 0,Y 209.078,Z 833.455,A -85,B 0,C 180,E1 11086.388,E2 11086.388} C_VEL
LIN {X 0,Y 208.258,Z 837.183,A -85,B 0,C 180,E1 11081.072,E2 11081.072} C_VEL
LIN {X 0,Y 208.151,Z 839.445,A -85,B 0,C 180,E1 11075.789,E2 11075.789} C_VEL
LIN {X 0,Y 208.232,Z 840.263,A -85,B 0,C 180,E1 11071.376,E2 11071.376} C_VEL
LIN {X 0,Y 208.194,Z 840.079,A -85,B 0,C 180,E1 11066.696,E2 11066.696} C_VEL
LIN {X 0,Y 208.145,Z 838.516,A -85,B 0,C 180,E1 11061.707,E2 11061.707} C_VEL
LIN {X 0,Y 208.529,Z 835.596,A -85,B 0,C 180,E1 11056.412,E2 11056.412} C_VEL
LIN {X 0,Y 209.926,Z 830.88,A -85,B 0,C 180,E1 11050.814,E2 11050.814} C_VEL
LIN {X 0,Y 212.834,Z 824.225,A -85,B 0,C 180,E1 11044.989,E2 11044.989} C_VEL
LIN {X 0,Y 217.136,Z 816.127,A -85,B 0,C 180,E1 11039.568,E2 11039.568} C_VEL
LIN {X 0,Y 223.017,Z 806.037,A -85,B 0,C 180,E1 11034.351,E2 11034.351} C_VEL
LIN {X 0,Y 230.052,Z 794.531,A -85,B 0,C 180,E1 11029.641,E2 11029.641} C_VEL
LIN {X 0,Y 237.962,Z 781.661,A -85,B 0,C 180,E1 11025.439,E2 11025.439} C_VEL
LIN {X 0,Y 246.581,Z 767.243,A -85,B 0,C 180,E1 11021.682,E2 11021.682} C_VEL
LIN {X 0,Y 255.358,Z 751.622,A -85,B 0,C 180,E1 11018.456,E2 11018.456} C_VEL
LIN {X 0,Y 264.145,Z 734.749,A -85,B 0,C 180,E1 11015.656,E2 11015.656} C_VEL
LIN {X 0,Y 272.676,Z 716.814,A -85,B 0,C 180,E1 11013.278,E2 11013.278} C_VEL
LIN {X 0,Y 280.736,Z 697.804,A -85,B 0,C 180,E1 11011.268,E2 11011.268} C_VEL
LIN {X 0,Y 287.712,Z 678.702,A -85,B 0,C 180,E1 11009.683,E2 11009.683} C_VEL
LIN {X 0,Y 293.812,Z 659.125,A -85,B 0,C 180,E1 11008.398,E2 11008.398} C_VEL
LIN {X 0,Y 299.207,Z 638.137,A -85,B 0,C 180,E1 11007.342,E2 11007.342} C_VEL
LIN {X 0,Y 303.553,Z 616.074,A -85,B 0,C 180,E1 11006.539,E2 11006.539} C_VEL
LIN {X 0,Y 306.348,Z 594.021,A -85,B 0,C 180,E1 11005.953,E2 11005.953} C_VEL
LIN {X 0,Y 319.751,Z 435.043,A -85,B 0,C 180,E1 11002.571,E2 11002.571} C_VEL
LIN {X 0,Y 314.095,Z 424.497,A -85,B 0,C 180,E1 10999.623,E2 10999.623} C_VEL
LIN {X 0,Y 309.214,Z 415.928,A -85,B 0,C 180,E1 10996.677,E2 10996.677} C_VEL
LIN {X 0,Y 304.517,Z 408.202,A -85,B 0,C 180,E1 10993.287,E2 10993.287} C_VEL
LIN {X 0,Y 301.179,Z 403.172,A -85,B 0,C 180,E1 10990.327,E2 10990.327} C_VEL
LIN {X 0,Y 298.548,Z 399.029,A -85,B 0,C 180,E1 10987.311,E2 10987.311} C_VEL
LIN {X 0,Y 295.501,Z 394.384,A -85,B 0,C 180,E1 10981.551,E2 10981.551} C_VEL
LIN {X 0,Y 294.854,Z 394.017,A -85,B 0,C 180,E1 10976.5,E2 10976.5} C_VEL
LIN {X 0,Y 295.271,Z 394.74,A -85,B 0,C 180,E1 10973.974,E2 10973.974} C_VEL
LIN {X 0,Y 297.839,Z 399.377,A -85,B 0,C 180,E1 10968.478,E2 10968.478} C_VEL
LIN {X 0,Y 300.372,Z 403.65,A -85,B 0,C 180,E1 10965.345,E2 10965.345} C_VEL
LIN {X 0,Y 303.313,Z 408.64,A -85,B 0,C 180,E1 10962.543,E2 10962.543} C_VEL
LIN {X 0,Y 307.417,Z 415.803,A -85,B 0,C 180,E1 10959.385,E2 10959.385} C_VEL
LIN {X 0,Y 311.661,Z 423.494,A -85,B 0,C 180,E1 10956.658,E2 10956.658} C_VEL
LIN {X 0,Y 317.085,Z 434.058,A -85,B 0,C 180,E1 10953.651,E2 10953.651} C_VEL
LIN {X 0,Y 318.43,Z 437.15,A -85,B 0,C 180,E1 10952.951,E2 10952.951} C_VEL
LIN {X 0,Y 305.593,Z 598.036,A -85,B 0,C 180,E1 10949.682,E2 10949.682} C_VEL
LIN {X 0,Y 302.368,Z 619.402,A -85,B 0,C 180,E1 10949.035,E2 10949.035} C_VEL
LIN {X 0,Y 298.046,Z 639.713,A -85,B 0,C 180,E1 10948.163,E2 10948.163} C_VEL
LIN {X 0,Y 292.258,Z 660.769,A -85,B 0,C 180,E1 10946.946,E2 10946.946} C_VEL
LIN {X 0,Y 286.102,Z 679.181,A -85,B 0,C 180,E1 10945.562,E2 10945.562} C_VEL
LIN {X 0,Y 278.775,Z 697.674,A -85,B 0,C 180,E1 10943.8,E2 10943.8} C_VEL
LIN {X 0,Y 270.736,Z 715.187,A -85,B 0,C 180,E1 10941.682,E2 10941.682} C_VEL
LIN {X 0,Y 262.529,Z 731.088,A -85,B 0,C 180,E1 10939.278,E2 10939.278} C_VEL
LIN {X 0,Y 253.927,Z 746.202,A -85,B 0,C 180,E1 10936.427,E2 10936.427} C_VEL
LIN {X 0,Y 245.457,Z 759.922,A -85,B 0,C 180,E1 10933.182,E2 10933.182} C_VEL
LIN {X 0,Y 236.853,Z 772.846,A -85,B 0,C 180,E1 10929.286,E2 10929.286} C_VEL
LIN {X 0,Y 229.344,Z 783.644,A -85,B 0,C 180,E1 10925.132,E2 10925.132} C_VEL
LIN {X 0,Y 222.353,Z 793.546,A -85,B 0,C 180,E1 10920.24,E2 10920.24} C_VEL
LIN {X 0,Y 216.852,Z 801.499,A -85,B 0,C 180,E1 10915.099,E2 10915.099} C_VEL
LIN {X 0,Y 212.689,Z 807.95,A -85,B 0,C 180,E1 10909.497,E2 10909.497} C_VEL
LIN {X 0,Y 210.067,Z 812.535,A -85,B 0,C 180,E1 10903.767,E2 10903.767} C_VEL
LIN {X 0,Y 208.796,Z 815.35,A -85,B 0,C 180,E1 10898.259,E2 10898.259} C_VEL
LIN {X 0,Y 208.353,Z 816.79,A -85,B 0,C 180,E1 10892.751,E2 10892.751} C_VEL
LIN {X 0,Y 208.33,Z 816.841,A -85,B 0,C 180,E1 10887.8,E2 10887.8} C_VEL
LIN {X 0,Y 208.712,Z 815.615,A -85,B 0,C 180,E1 10882.291,E2 10882.291} C_VEL
LIN {X 0,Y 209.872,Z 813.002,A -85,B 0,C 180,E1 10876.781,E2 10876.781} C_VEL
LIN {X 0,Y 212.324,Z 808.541,A -85,B 0,C 180,E1 10871.039,E2 10871.039} C_VEL
LIN {X 0,Y 216.09,Z 802.665,A -85,B 0,C 180,E1 10865.682,E2 10865.682} C_VEL
LIN {X 0,Y 221.352,Z 795.071,A -85,B 0,C 180,E1 10860.505,E2 10860.505} C_VEL
LIN {X 0,Y 227.732,Z 786.1,A -85,B 0,C 180,E1 10855.808,E2 10855.808} C_VEL
LIN {X 0,Y 235.414,Z 775.074,A -85,B 0,C 180,E1 10851.367,E2 10851.367} C_VEL
LIN {X 0,Y 243.323,Z 763.264,A -85,B 0,C 180,E1 10847.632,E2 10847.632} C_VEL
LIN {X 0,Y 252.147,Z 749.307,A -85,B 0,C 180,E1 10844.134,E2 10844.134} C_VEL
LIN {X 0,Y 260.623,Z 734.82,A -85,B 0,C 180,E1 10841.243,E2 10841.243} C_VEL
LIN {X 0,Y 269.069,Z 718.865,A -85,B 0,C 180,E1 10838.709,E2 10838.709} C_VEL
